LIN {X 0,Y 282.831,Z 361.895,A -85,B 0,C 180,E1 -17098.576,E2 -17098.576} C_VEL
LIN {X 0,Y 282.658,Z 360.951,A -85,B 0,C 180,E1 -17100,E2 -17100} C_VEL
LIN {X 0,Y 282.587,Z 359.569,A -85,B 0,C 180,E1 -17101.425,E2 -17101.425} C_VEL
LIN {X 0,Y 282.639,Z 356.738,A -85,B 0,C 180,E1 -17103.564,E2 -17103.564} C_VEL
LIN {X 0,Y 282.765,Z 351.895,A -85,B 0,C 180,E1 -17106.179,E2 -17106.179} C_VEL
LIN {X 0,Y 283.123,Z 346.036,A -85,B 0,C 180,E1 -17108.566,E2 -17108.566} C_VEL
LIN {X 0,Y 283.616,Z 339.368,A -85,B 0,C 180,E1 -17110.711,E2 -17110.711} C_VEL
LIN {X 0,Y 284.287,Z 331.159,A -85,B 0,C 180,E1 -17112.856,E2 -17112.856} C_VEL
LIN {X 0,Y 285.11,Z 322.916,A -85,B 0,C 180,E1 -17114.635,E2 -17114.635} C_VEL
LIN {X 0,Y 285.821,Z 314.704,A -85,B 0,C 180,E1 -17116.129,E2 -17116.129} C_VEL
LIN {X 0,Y 286.898,Z 303.457,A -85,B 0,C 180,E1 -17117.831,E2 -17117.831} C_VEL
LIN {X 0,Y 288.151,Z 290.351,A -85,B 0,C 180,E1 -17119.41,E2 -17119.41} C_VEL
LIN {X 0,Y 288.308,Z 286.867,A -85,B 0,C 180,E1 -17119.769,E2 -17119.769} C_VEL
LIN {X 0,Y 286.028,Z 274.318,A -85,B 0,C 180,E1 -17120.979,E2 -17120.979} C_VEL
LIN {X 0,Y 283.378,Z 259.454,A -85,B 0,C 180,E1 -17122.077,E2 -17122.077} C_VEL
LIN {X 0,Y 282.903,Z 256.645,A -85,B 0,C 180,E1 -17122.25,E2 -17122.25} C_VEL
LIN {X 0,Y 283.071,Z 253.228,A -85,B 0,C 180,E1 -17126.148,E2 -17126.148} C_VEL
LIN {X 0,Y 283.439,Z 253.178,A -85,B 0,C 180,E1 -17129.79,E2 -17129.79} C_VEL
LIN {X 0,Y 283.84,Z 253.128,A -85,B 0,C 180,E1 -17133.007,E2 -17133.007} C_VEL
LIN {X 0,Y 284.182,Z 253.083,A -85,B 0,C 180,E1 -17136.409,E2 -17136.409} C_VEL
LIN {X 0,Y 284.308,Z 253.067,A -85,B 0,C 180,E1 -17139.995,E2 -17139.995} C_VEL
LIN {X 0,Y 284.248,Z 253.076,A -85,B 0,C 180,E1 -17144.19,E2 -17144.19} C_VEL
LIN {X 0,Y 284.243,Z 253.076,A -85,B 0,C 180,E1 -17148.119,E2 -17148.119} C_VEL
LIN {X 0,Y 284.311,Z 253.069,A -85,B 0,C 180,E1 -17152.282,E2 -17152.282} C_VEL
LIN {X 0,Y 284.31,Z 253.069,A -85,B 0,C 180,E1 -17155.35,E2 -17155.35} C_VEL
LIN {X 0,Y 284.29,Z 253.074,A -85,B 0,C 180,E1 -17158.725,E2 -17158.725} C_VEL
LIN {X 0,Y 284.294,Z 253.071,A -85,B 0,C 180,E1 -17161.985,E2 -17161.985} C_VEL
LIN {X 0,Y 284.329,Z 253.068,A -85,B 0,C 180,E1 -17166.145,E2 -17166.145} C_VEL
LIN {X 0,Y 284.391,Z 253.059,A -85,B 0,C 180,E1 -17169.898,E2 -17169.898} C_VEL
LIN {X 0,Y 284.496,Z 253.047,A -85,B 0,C 180,E1 -17174.459,E2 -17174.459} C_VEL
LIN {X 0,Y 284.486,Z 253.048,A -85,B 0,C 180,E1 -17178.601,E2 -17178.601} C_VEL
LIN {X 0,Y 284.611,Z 253.033,A -85,B 0,C 180,E1 -17181.479,E2 -17181.479} C_VEL
LIN {X 0,Y 284.568,Z 253.038,A -85,B 0,C 180,E1 -17184.33,E2 -17184.33} C_VEL
LIN {X 0,Y 284.844,Z 253.003,A -85,B 0,C 180,E1 -17188.586,E2 -17188.586} C_VEL
LIN {X 0,Y 284.839,Z 253.007,A -85,B 0,C 180,E1 -17191.414,E2 -17191.414} C_VEL
LIN {X 0,Y 284.646,Z 253.052,A -85,B 0,C 180,E1 -17193.007,E2 -17193.007} C_VEL
LIN {X 0,Y 284.818,Z 258.793,A -85,B 0,C 180,E1 -17196.375,E2 -17196.375} C_VEL
LIN {X 0,Y 284.369,Z 266.259,A -85,B 0,C 180,E1 -17200.682,E2 -17200.682} C_VEL
LIN {X 0,Y 284.094,Z 272.577,A -85,B 0,C 180,E1 -17204.323,E2 -17204.323} C_VEL
LIN {X 0,Y 283.88,Z 279.623,A -85,B 0,C 180,E1 -17208.307,E2 -17208.307} C_VEL
LIN {X 0,Y 285.728,Z 289.55,A -85,B 0,C 180,E1 -17208.927,E2 -17208.927} C_VEL
LIN {X 0,Y 287.481,Z 300.318,A -85,B 0,C 180,E1 -17209.828,E2 -17209.828} C_VEL
LIN {X 0,Y 288.186,Z 306.947,A -85,B 0,C 180,E1 -17210.522,E2 -17210.522} C_VEL
LIN {X 0,Y 287.358,Z 316.725,A -85,B 0,C 180,E1 -17211.661,E2 -17211.661} C_VEL
LIN {X 0,Y 286.342,Z 326.267,A -85,B 0,C 180,E1 -17213.123,E2 -17213.123} C_VEL
LIN {X 0,Y 285.604,Z 333.152,A -85,B 0,C 180,E1 -17214.427,E2 -17214.427} C_VEL
LIN {X 0,Y 285.015,Z 338.231,A -85,B 0,C 180,E1 -17215.564,E2 -17215.564} C_VEL
LIN {X 0,Y 284.307,Z 344.063,A -85,B 0,C 180,E1 -17217.137,E2 -17217.137} C_VEL
LIN {X 0,Y 283.686,Z 349.285,A -85,B 0,C 180,E1 -17218.887,E2 -17218.887} C_VEL
LIN {X 0,Y 283.192,Z 353.281,A -85,B 0,C 180,E1 -17220.58,E2 -17220.58} C_VEL
LIN {X 0,Y 282.836,Z 356.48,A -85,B 0,C 180,E1 -17222.344,E2 -17222.344} C_VEL
LIN {X 0,Y 282.69,Z 357.695,A -85,B 0,C 180,E1 -17223.158,E2 -17223.158} C_VEL
LIN {X 0,Y 282.49,Z 359.603,A -85,B 0,C 180,E1 -17224.905,E2 -17224.905} C_VEL
LIN {X 0,Y 282.397,Z 360.883,A -85,B 0,C 180,E1 -17227.213,E2 -17227.213} C_VEL
LIN {X 0,Y 282.468,Z 361.102,A -85,B 0,C 180,E1 -17228.464,E2 -17228.464} C_VEL
LIN {X 0,Y 282.717,Z 360.662,A -85,B 0,C 180,E1 -17230.265,E2 -17230.265} C_VEL
LIN {X 0,Y 283.098,Z 359.387,A -85,B 0,C 180,E1 -17232.089,E2 -17232.089} C_VEL
LIN {X 0,Y 283.686,Z 356.998,A -85,B 0,C 180,E1 -17234.074,E2 -17234.074} C_VEL
LIN {X 0,Y 284.532,Z 353.138,A -85,B 0,C 180,E1 -17236.242,E2 -17236.242} C_VEL
LIN {X 0,Y 285.66,Z 347.925,A -85,B 0,C 180,E1 -17238.373,E2 -17238.373} C_VEL
LIN {X 0,Y 286.946,Z 340.998,A -85,B 0,C 180,E1 -17240.446,E2 -17240.446} C_VEL
LIN {X 0,Y 288.222,Z 334.615,A -85,B 0,C 180,E1 -17241.948,E2 -17241.948} C_VEL
LIN {X 0,Y 289.382,Z 327.787,A -85,B 0,C 180,E1 -17243.268,E2 -17243.268} C_VEL
LIN {X 0,Y 290.809,Z 318.256,A -85,B 0,C 180,E1 -17244.757,E2 -17244.757} C_VEL
LIN {X 0,Y 291.63,Z 311.075,A -85,B 0,C 180,E1 -17245.652,E2 -17245.652} C_VEL
LIN {X 0,Y 290.183,Z 300.685,A -85,B 0,C 180,E1 -17246.889,E2 -17246.889} C_VEL
LIN {X 0,Y 288.063,Z 291.312,A -85,B 0,C 180,E1 -17247.848,E2 -17247.848} C_VEL
LIN {X 0,Y 285.192,Z 281.882,A -85,B 0,C 180,E1 -17248.68,E2 -17248.68} C_VEL
LIN {X 0,Y 284.996,Z 280.806,A -85,B 0,C 180,E1 -17248.811,E2 -17248.811} C_VEL
LIN {X 0,Y 285.473,Z 273.627,A -85,B 0,C 180,E1 -17253.077,E2 -17253.077} C_VEL
LIN {X 0,Y 285.948,Z 266.001,A -85,B 0,C 180,E1 -17257.607,E2 -17257.607} C_VEL
LIN {X 0,Y 286.031,Z 262.289,A -85,B 0,C 180,E1 -17259.88,E2 -17259.88} C_VEL
LIN {X 0,Y 285.367,Z 257.623,A -85,B 0,C 180,E1 -17262.81,E2 -17262.81} C_VEL
LIN {X 0,Y 284.5,Z 253.05,A -85,B 0,C 180,E1 -17265.88,E2 -17265.88} C_VEL
LIN {X 0,Y 284.521,Z 253.047,A -85,B 0,C 180,E1 -17270.046,E2 -17270.046} C_VEL
LIN {X 0,Y 284.662,Z 253.027,A -85,B 0,C 180,E1 -17272.909,E2 -17272.909} C_VEL
LIN {X 0,Y 284.554,Z 253.037,A -85,B 0,C 180,E1 -17276.166,E2 -17276.166} C_VEL
LIN {X 0,Y 284.035,Z 253.105,A -85,B 0,C 180,E1 -17277.35,E2 -17277.35} C_VEL
LIN {X 0,Y 281.309,Z 253.443,A -85,B 0,C 180,E1 -17279.282,E2 -17279.282} C_VEL
LIN {X 0,Y 278.895,Z 253.747,A -85,B 0,C 180,E1 -17280.851,E2 -17280.851} C_VEL
LIN {X 0,Y 277.82,Z 253.879,A -85,B 0,C 180,E1 -17282.066,E2 -17282.066} C_VEL
LIN {X 0,Y 277.716,Z 253.89,A -85,B 0,C 180,E1 -17282.477,E2 -17282.477} C_VEL
LIN {X 0,Y 277.613,Z 253.907,A -85,B 0,C 180,E1 -17287.272,E2 -17287.272} C_VEL
LIN {X 0,Y 277.462,Z 253.924,A -85,B 0,C 180,E1 -17290.213,E2 -17290.213} C_VEL
LIN {X 0,Y 277.436,Z 253.928,A -85,B 0,C 180,E1 -17294.674,E2 -17294.674} C_VEL
LIN {X 0,Y 277.346,Z 253.935,A -85,B 0,C 180,E1 -17299.234,E2 -17299.234} C_VEL
LIN {X 0,Y 277.293,Z 253.941,A -85,B 0,C 180,E1 -17304.158,E2 -17304.158} C_VEL
LIN {X 0,Y 277.327,Z 253.938,A -85,B 0,C 180,E1 -17307.505,E2 -17307.505} C_VEL
LIN {X 0,Y 277.273,Z 253.947,A -85,B 0,C 180,E1 -17310.481,E2 -17310.481} C_VEL
LIN {X 0,Y 277.248,Z 253.949,A -85,B 0,C 180,E1 -17313.896,E2 -17313.896} C_VEL
LIN {X 0,Y 277.273,Z 253.943,A -85,B 0,C 180,E1 -17317.468,E2 -17317.468} C_VEL
LIN {X 0,Y 277.216,Z 253.954,A -85,B 0,C 180,E1 -17321.235,E2 -17321.235} C_VEL
LIN {X 0,Y 277.356,Z 254.102,A -85,B 0,C 180,E1 -17324.424,E2 -17324.424} C_VEL
LIN {X 0,Y 278.44,Z 259.918,A -85,B 0,C 180,E1 -17328.985,E2 -17328.985} C_VEL
LIN {X 0,Y 279.116,Z 264.08,A -85,B 0,C 180,E1 -17332.105,E2 -17332.105} C_VEL
LIN {X 0,Y 279.095,Z 267.562,A -85,B 0,C 180,E1 -17334.608,E2 -17334.608} C_VEL
LIN {X 0,Y 278.184,Z 272.378,A -85,B 0,C 180,E1 -17337.958,E2 -17337.958} C_VEL
LIN {X 0,Y 277.416,Z 277.12,A -85,B 0,C 180,E1 -17341.227,E2 -17341.227} C_VEL
LIN {X 0,Y 276.912,Z 281.064,A -85,B 0,C 180,E1 -17343.834,E2 -17343.834} C_VEL
LIN {X 0,Y 278.169,Z 295.048,A -85,B 0,C 180,E1 -17346.748,E2 -17346.748} C_VEL
LIN {X 0,Y 278.48,Z 299.439,A -85,B 0,C 180,E1 -17347.56,E2 -17347.56} C_VEL
LIN {X 0,Y 279.824,Z 307.988,A -85,B 0,C 180,E1 -17348.027,E2 -17348.027} C_VEL
LIN {X 0,Y 280.79,Z 317.875,A -85,B 0,C 180,E1 -17348.666,E2 -17348.666} C_VEL
LIN {X 0,Y 281.623,Z 328.142,A -85,B 0,C 180,E1 -17349.551,E2 -17349.551} C_VEL
LIN {X 0,Y 281.925,Z 335.562,A -85,B 0,C 180,E1 -17350.334,E2 -17350.334} C_VEL
LIN {X 0,Y 280.797,Z 346.088,A -85,B 0,C 180,E1 -17351.58,E2 -17351.58} C_VEL
LIN {X 0,Y 279.658,Z 354.16,A -85,B 0,C 180,E1 -17352.808,E2 -17352.808} C_VEL
LIN {X 0,Y 278.667,Z 361.864,A -85,B 0,C 180,E1 -17354.269,E2 -17354.269} C_VEL
LIN {X 0,Y 277.805,Z 368.163,A -85,B 0,C 180,E1 -17355.72,E2 -17355.72} C_VEL
LIN {X 0,Y 276.985,Z 373.425,A -85,B 0,C 180,E1 -17357.173,E2 -17357.173} C_VEL
LIN {X 0,Y 276.277,Z 378.801,A -85,B 0,C 180,E1 -17359.001,E2 -17359.001} C_VEL
LIN {X 0,Y 275.896,Z 382.288,A -85,B 0,C 180,E1 -17360.469,E2 -17360.469} C_VEL
LIN {X 0,Y 275.532,Z 386.34,A -85,B 0,C 180,E1 -17362.673,E2 -17362.673} C_VEL
LIN {X 0,Y 275.44,Z 388.507,A -85,B 0,C 180,E1 -17364.331,E2 -17364.331} C_VEL
LIN {X 0,Y 275.41,Z 389.721,A -85,B 0,C 180,E1 -17365.61,E2 -17365.61} C_VEL
LIN {X 0,Y 275.499,Z 390.664,A -85,B 0,C 180,E1 -17367.076,E2 -17367.076} C_VEL
LIN {X 0,Y 275.55,Z 391.055,A -85,B 0,C 180,E1 -17368.539,E2 -17368.539} C_VEL
LIN {X 0,Y 275.637,Z 390.67,A -85,B 0,C 180,E1 -17371.461,E2 -17371.461} C_VEL
LIN {X 0,Y 275.355,Z 391.344,A -85,B 0,C 180,E1 -17374.392,E2 -17374.392} C_VEL
LIN {X 0,Y 275.454,Z 390.474,A -85,B 0,C 180,E1 -17377.33,E2 -17377.33} C_VEL
LIN {X 0,Y 275.722,Z 389.465,A -85,B 0,C 180,E1 -17378.797,E2 -17378.797} C_VEL
LIN {X 0,Y 276.728,Z 386.251,A -85,B 0,C 180,E1 -17381.723,E2 -17381.723} C_VEL
LIN {X 0,Y 277.919,Z 382.837,A -85,B 0,C 180,E1 -17383.901,E2 -17383.901} C_VEL
LIN {X 0,Y 280.452,Z 376.813,A -85,B 0,C 180,E1 -17386.75,E2 -17386.75} C_VEL
LIN {X 0,Y 282.55,Z 371.143,A -85,B 0,C 180,E1 -17388.866,E2 -17388.866} C_VEL
LIN {X 0,Y 285.852,Z 363.067,A -85,B 0,C 180,E1 -17391.263,E2 -17391.263} C_VEL
LIN {X 0,Y 289.91,Z 353.174,A -85,B 0,C 180,E1 -17393.578,E2 -17393.578} C_VEL
LIN {X 0,Y 293.011,Z 344.832,A -85,B 0,C 180,E1 -17395.198,E2 -17395.198} C_VEL
LIN {X 0,Y 294.489,Z 337.714,A -85,B 0,C 180,E1 -17396.582,E2 -17396.582} C_VEL
LIN {X 0,Y 295.186,Z 329.455,A -85,B 0,C 180,E1 -17398.246,E2 -17398.246} C_VEL
LIN {X 0,Y 294.967,Z 319.929,A -85,B 0,C 180,E1 -17400.266,E2 -17400.266} C_VEL
LIN {X 0,Y 294.401,Z 313.67,A -85,B 0,C 180,E1 -17401.681,E2 -17401.681} C_VEL
LIN {X 0,Y 292.788,Z 303.44,A -85,B 0,C 180,E1 -17404.3,E2 -17404.3} C_VEL
LIN {X 0,Y 292.15,Z 300.019,A -85,B 0,C 180,E1 -17405.265,E2 -17405.265} C_VEL
LIN {X 0,Y 290.757,Z 294.362,A -85,B 0,C 180,E1 -17407.178,E2 -17407.178} C_VEL
LIN {X 0,Y 289.417,Z 289.757,A -85,B 0,C 180,E1 -17409.152,E2 -17409.152} C_VEL
LIN {X 0,Y 288.8,Z 287.91,A -85,B 0,C 180,E1 -17410.144,E2 -17410.144} C_VEL
LIN {X 0,Y 287.153,Z 284.531,A -85,B 0,C 180,E1 -17413.259,E2 -17413.259} C_VEL
LIN {X 0,Y 286.793,Z 283.133,A -85,B 0,C 180,E1 -17415.289,E2 -17415.289} C_VEL
LIN {X 0,Y 286.896,Z 282.566,A -85,B 0,C 180,E1 -17417.299,E2 -17417.299} C_VEL
LIN {X 0,Y 288.338,Z 282.932,A -85,B 0,C 180,E1 -17420.674,E2 -17420.674} C_VEL
LIN {X 0,Y 288.675,Z 283.13,A -85,B 0,C 180,E1 -17421.176,E2 -17421.176} C_VEL
LIN {X 0,Y 291.63,Z 287.665,A -85,B 0,C 180,E1 -17425.022,E2 -17425.022} C_VEL
LIN {X 0,Y 294.048,Z 292.584,A -85,B 0,C 180,E1 -17427.557,E2 -17427.557} C_VEL
LIN {X 0,Y 296.068,Z 297.264,A -85,B 0,C 180,E1 -17429.494,E2 -17429.494} C_VEL
LIN {X 0,Y 298.512,Z 305.114,A -85,B 0,C 180,E1 -17432.111,E2 -17432.111} C_VEL
LIN {X 0,Y 299.925,Z 313.163,A -85,B 0,C 180,E1 -17434.397,E2 -17434.397} C_VEL
LIN {X 0,Y 300.069,Z 314.428,A -85,B 0,C 180,E1 -17434.738,E2 -17434.738} C_VEL
LIN {X 0,Y 299.8,Z 315.956,A -85,B 0,C 180,E1 -17435.042,E2 -17435.042} C_VEL
LIN {X 0,Y 295.732,Z 326.426,A -85,B 0,C 180,E1 -17436.914,E2 -17436.914} C_VEL
LIN {X 0,Y 292.089,Z 335.102,A -85,B 0,C 180,E1 -17438.844,E2 -17438.844} C_VEL
LIN {X 0,Y 288.331,Z 343.318,A -85,B 0,C 180,E1 -17441.158,E2 -17441.158} C_VEL
LIN {X 0,Y 285.081,Z 349.926,A -85,B 0,C 180,E1 -17443.531,E2 -17443.531} C_VEL
LIN {X 0,Y 282.003,Z 355.656,A -85,B 0,C 180,E1 -17446.305,E2 -17446.305} C_VEL
LIN {X 0,Y 280.101,Z 358.853,A -85,B 0,C 180,E1 -17448.421,E2 -17448.421} C_VEL
LIN {X 0,Y 278.918,Z 360.509,A -85,B 0,C 180,E1 -17449.841,E2 -17449.841} C_VEL
LIN {X 0,Y 278.251,Z 361.729,A -85,B 0,C 180,E1 -17451.284,E2 -17451.284} C_VEL
LIN {X 0,Y 277.048,Z 363.021,A -85,B 0,C 180,E1 -17454.176,E2 -17454.176} C_VEL
LIN {X 0,Y 276.62,Z 363.112,A -85,B 0,C 180,E1 -17455.629,E2 -17455.629} C_VEL
LIN {X 0,Y 276.092,Z 362.846,A -85,B 0,C 180,E1 -17457.082,E2 -17457.082} C_VEL
LIN {X 0,Y 275.739,Z 362.169,A -85,B 0,C 180,E1 -17458.54,E2 -17458.54} C_VEL
LIN {X 0,Y 275.502,Z 359.588,A -85,B 0,C 180,E1 -17461.462,E2 -17461.462} C_VEL
LIN {X 0,Y 275.554,Z 356.575,A -85,B 0,C 180,E1 -17463.656,E2 -17463.656} C_VEL
LIN {X 0,Y 275.66,Z 352.015,A -85,B 0,C 180,E1 -17466.109,E2 -17466.109} C_VEL
LIN {X 0,Y 275.956,Z 347.388,A -85,B 0,C 180,E1 -17468.052,E2 -17468.052} C_VEL
LIN {X 0,Y 276.41,Z 340.976,A -85,B 0,C 180,E1 -17470.252,E2 -17470.252} C_VEL
LIN {X 0,Y 277.019,Z 333.069,A -85,B 0,C 180,E1 -17472.454,E2 -17472.454} C_VEL
LIN {X 0,Y 278,Z 323.322,A -85,B 0,C 180,E1 -17474.644,E2 -17474.644} C_VEL
LIN {X 0,Y 278.778,Z 314.188,A -85,B 0,C 180,E1 -17476.341,E2 -17476.341} C_VEL
LIN {X 0,Y 279.941,Z 302.606,A -85,B 0,C 180,E1 -17478.1,E2 -17478.1} C_VEL
LIN {X 0,Y 281.058,Z 290.91,A -85,B 0,C 180,E1 -17479.539,E2 -17479.539} C_VEL
LIN {X 0,Y 281.219,Z 287.457,A -85,B 0,C 180,E1 -17479.908,E2 -17479.908} C_VEL
LIN {X 0,Y 278.876,Z 274.615,A -85,B 0,C 180,E1 -17481.18,E2 -17481.18} C_VEL
LIN {X 0,Y 276.275,Z 259.963,A -85,B 0,C 180,E1 -17482.291,E2 -17482.291} C_VEL
LIN {X 0,Y 275.804,Z 257.028,A -85,B 0,C 180,E1 -17482.472,E2 -17482.472} C_VEL
LIN {X 0,Y 275.996,Z 254.109,A -85,B 0,C 180,E1 -17486.05,E2 -17486.05} C_VEL
LIN {X 0,Y 276.468,Z 254.045,A -85,B 0,C 180,E1 -17490.559,E2 -17490.559} C_VEL
LIN {X 0,Y 276.896,Z 253.99,A -85,B 0,C 180,E1 -17493.945,E2 -17493.945} C_VEL
LIN {X 0,Y 277.195,Z 253.957,A -85,B 0,C 180,E1 -17497.481,E2 -17497.481} C_VEL
LIN {X 0,Y 277.213,Z 253.955,A -85,B 0,C 180,E1 -17501.236,E2 -17501.236} C_VEL
LIN {X 0,Y 277.204,Z 253.956,A -85,B 0,C 180,E1 -17505.226,E2 -17505.226} C_VEL
LIN {X 0,Y 277.2,Z 253.955,A -85,B 0,C 180,E1 -17509.518,E2 -17509.518} C_VEL
LIN {X 0,Y 277.257,Z 253.949,A -85,B 0,C 180,E1 -17512.529,E2 -17512.529} C_VEL
LIN {X 0,Y 277.249,Z 253.949,A -85,B 0,C 180,E1 -17516.104,E2 -17516.104} C_VEL
LIN {X 0,Y 277.265,Z 253.945,A -85,B 0,C 180,E1 -17519.538,E2 -17519.538} C_VEL
LIN {X 0,Y 277.309,Z 253.942,A -85,B 0,C 180,E1 -17522.858,E2 -17522.858} C_VEL
LIN {X 0,Y 277.29,Z 253.944,A -85,B 0,C 180,E1 -17526.076,E2 -17526.076} C_VEL
LIN {X 0,Y 277.348,Z 253.935,A -85,B 0,C 180,E1 -17530.766,E2 -17530.766} C_VEL
LIN {X 0,Y 277.438,Z 253.924,A -85,B 0,C 180,E1 -17535.326,E2 -17535.326} C_VEL
LIN {X 0,Y 277.461,Z 253.925,A -85,B 0,C 180,E1 -17539.787,E2 -17539.787} C_VEL
LIN {X 0,Y 277.602,Z 253.905,A -85,B 0,C 180,E1 -17542.727,E2 -17542.727} C_VEL
LIN {X 0,Y 277.81,Z 253.879,A -85,B 0,C 180,E1 -17548.55,E2 -17548.55} C_VEL
LIN {X 0,Y 277.719,Z 253.892,A -85,B 0,C 180,E1 -17552.175,E2 -17552.175} C_VEL
LIN {X 0,Y 277.664,Z 254.036,A -85,B 0,C 180,E1 -17552.811,E2 -17552.811} C_VEL
LIN {X 0,Y 277.811,Z 259.03,A -85,B 0,C 180,E1 -17555.808,E2 -17555.808} C_VEL
LIN {X 0,Y 277.393,Z 266.586,A -85,B 0,C 180,E1 -17560.215,E2 -17560.215} C_VEL
LIN {X 0,Y 277.094,Z 272.975,A -85,B 0,C 180,E1 -17563.943,E2 -17563.943} C_VEL
LIN {X 0,Y 276.858,Z 279.85,A -85,B 0,C 180,E1 -17567.926,E2 -17567.926} C_VEL
LIN {X 0,Y 278.693,Z 289.804,A -85,B 0,C 180,E1 -17568.564,E2 -17568.564} C_VEL
LIN {X 0,Y 280.318,Z 299.627,A -85,B 0,C 180,E1 -17569.402,E2 -17569.402} C_VEL
LIN {X 0,Y 281.216,Z 306.242,A -85,B 0,C 180,E1 -17570.098,E2 -17570.098} C_VEL
LIN {X 0,Y 280.592,Z 314.904,A -85,B 0,C 180,E1 -17571.103,E2 -17571.103} C_VEL
LIN {X 0,Y 279.567,Z 324.771,A -85,B 0,C 180,E1 -17572.542,E2 -17572.542} C_VEL
LIN {X 0,Y 278.675,Z 332.941,A -85,B 0,C 180,E1 -17574.09,E2 -17574.09} C_VEL
LIN {X 0,Y 277.953,Z 338.903,A -85,B 0,C 180,E1 -17575.457,E2 -17575.457} C_VEL
LIN {X 0,Y 277.184,Z 344.955,A -85,B 0,C 180,E1 -17577.154,E2 -17577.154} C_VEL
LIN {X 0,Y 276.581,Z 349.874,A -85,B 0,C 180,E1 -17578.868,E2 -17578.868} C_VEL
LIN {X 0,Y 276.11,Z 353.826,A -85,B 0,C 180,E1 -17580.602,E2 -17580.602} C_VEL
LIN {X 0,Y 275.666,Z 357.483,A -85,B 0,C 180,E1 -17582.719,E2 -17582.719} C_VEL
LIN {X 0,Y 275.358,Z 360.186,A -85,B 0,C 180,E1 -17585.24,E2 -17585.24} C_VEL
LIN {X 0,Y 275.335,Z 361.392,A -85,B 0,C 180,E1 -17587.778,E2 -17587.778} C_VEL
LIN {X 0,Y 275.609,Z 361.227,A -85,B 0,C 180,E1 -17590.093,E2 -17590.093} C_VEL
LIN {X 0,Y 276.131,Z 359.671,A -85,B 0,C 180,E1 -17592.43,E2 -17592.43} C_VEL
LIN {X 0,Y 276.83,Z 356.888,A -85,B 0,C 180,E1 -17594.696,E2 -17594.696} C_VEL
LIN {X 0,Y 277.884,Z 352.329,A -85,B 0,C 180,E1 -17597.176,E2 -17597.176} C_VEL
LIN {X 0,Y 278.989,Z 347.362,A -85,B 0,C 180,E1 -17599.089,E2 -17599.089} C_VEL
LIN {X 0,Y 280.262,Z 340.907,A -85,B 0,C 180,E1 -17601.021,E2 -17601.021} C_VEL
LIN {X 0,Y 281.709,Z 333.87,A -85,B 0,C 180,E1 -17602.683,E2 -17602.683} C_VEL
LIN {X 0,Y 283.337,Z 324.577,A -85,B 0,C 180,E1 -17604.41,E2 -17604.41} C_VEL
LIN {X 0,Y 284.59,Z 316.244,A -85,B 0,C 180,E1 -17605.61,E2 -17605.61} C_VEL
LIN {X 0,Y 284.925,Z 311.04,A -85,B 0,C 180,E1 -17606.29,E2 -17606.29} C_VEL
LIN {X 0,Y 283.475,Z 301.24,A -85,B 0,C 180,E1 -17607.497,E2 -17607.497} C_VEL
LIN {X 0,Y 281.225,Z 291.571,A -85,B 0,C 180,E1 -17608.526,E2 -17608.526} C_VEL
LIN {X 0,Y 278.25,Z 281.865,A -85,B 0,C 180,E1 -17609.426,E2 -17609.426} C_VEL
LIN {X 0,Y 278.135,Z 281.189,A -85,B 0,C 180,E1 -17609.528,E2 -17609.528} C_VEL
LIN {X 0,Y 278.519,Z 275.466,A -85,B 0,C 180,E1 -17612.986,E2 -17612.986} C_VEL
LIN {X 0,Y 279.099,Z 267.527,A -85,B 0,C 180,E1 -17617.807,E2 -17617.807} C_VEL
LIN {X 0,Y 279.158,Z 263.819,A -85,B 0,C 180,E1 -17620.131,E2 -17620.131} C_VEL
LIN {X 0,Y 278.689,Z 260.323,A -85,B 0,C 180,E1 -17622.385,E2 -17622.385} C_VEL
LIN {X 0,Y 277.638,Z 254.834,A -85,B 0,C 180,E1 -17626.085,E2 -17626.085} C_VEL
LIN {X 0,Y 277.431,Z 253.926,A -85,B 0,C 180,E1 -17626.821,E2 -17626.821} C_VEL
LIN {X 0,Y 277.599,Z 253.908,A -85,B 0,C 180,E1 -17631.263,E2 -17631.263} C_VEL
LIN {X 0,Y 277.553,Z 253.912,A -85,B 0,C 180,E1 -17634.187,E2 -17634.187} C_VEL
LIN {X 0,Y 277.822,Z 253.88,A -85,B 0,C 180,E1 -17638.55,E2 -17638.55} C_VEL
LIN {X 0,Y 277.822,Z 253.877,A -85,B 0,C 180,E1 -17641.449,E2 -17641.449} C_VEL
LIN {X 0,Y 277.716,Z 253.89,A -85,B 0,C 180,E1 -17642.477,E2 -17642.477} C_VEL
LIN {X 0,Y 276.988,Z 253.984,A -85,B 0,C 180,E1 -17643.686,E2 -17643.686} C_VEL
LIN {X 0,Y 274.06,Z 254.346,A -85,B 0,C 180,E1 -17645.654,E2 -17645.654} C_VEL
LIN {X 0,Y 271.62,Z 254.653,A -85,B 0,C 180,E1 -17647.253,E2 -17647.253} C_VEL
LIN {X 0,Y 270.598,Z 254.776,A -85,B 0,C 180,E1 -17648.494,E2 -17648.494} C_VEL
LIN {X 0,Y 270.527,Z 254.786,A -85,B 0,C 180,E1 -17648.914,E2 -17648.914} C_VEL
LIN {X 0,Y 270.361,Z 254.804,A -85,B 0,C 180,E1 -17653.53,E2 -17653.53} C_VEL
LIN {X 0,Y 270.356,Z 254.805,A -85,B 0,C 180,E1 -17656.615,E2 -17656.615} C_VEL
LIN {X 0,Y 270.292,Z 254.816,A -85,B 0,C 180,E1 -17660.601,E2 -17660.601} C_VEL
LIN {X 0,Y 270.239,Z 254.821,A -85,B 0,C 180,E1 -17664.589,E2 -17664.589} C_VEL
LIN {X 0,Y 270.273,Z 254.82,A -85,B 0,C 180,E1 -17667.908,E2 -17667.908} C_VEL
LIN {X 0,Y 270.185,Z 254.828,A -85,B 0,C 180,E1 -17671.348,E2 -17671.348} C_VEL
LIN {X 0,Y 270.203,Z 254.823,A -85,B 0,C 180,E1 -17674.905,E2 -17674.905} C_VEL
LIN {X 0,Y 270.198,Z 254.828,A -85,B 0,C 180,E1 -17678.71,E2 -17678.71} C_VEL
LIN {X 0,Y 270.219,Z 254.827,A -85,B 0,C 180,E1 -17683.261,E2 -17683.261} C_VEL
LIN {X 0,Y 270.321,Z 255.015,A -85,B 0,C 180,E1 -17684.4,E2 -17684.4} C_VEL
LIN {X 0,Y 271.317,Z 260.334,A -85,B 0,C 180,E1 -17688.694,E2 -17688.694} C_VEL
LIN {X 0,Y 272.101,Z 265.284,A -85,B 0,C 180,E1 -17692.501,E2 -17692.501} C_VEL
LIN {X 0,Y 272.043,Z 267.943,A -85,B 0,C 180,E1 -17694.46,E2 -17694.46} C_VEL
LIN {X 0,Y 271.111,Z 272.74,A -85,B 0,C 180,E1 -17697.899,E2 -17697.899} C_VEL
LIN {X 0,Y 270.078,Z 279.195,A -85,B 0,C 180,E1 -17702.448,E2 -17702.448} C_VEL
LIN {X 0,Y 271.191,Z 292.709,A -85,B 0,C 180,E1 -17705.503,E2 -17705.503} C_VEL
LIN {X 0,Y 271.702,Z 299.153,A -85,B 0,C 180,E1 -17706.804,E2 -17706.804} C_VEL
LIN {X 0,Y 273.014,Z 305.084,A -85,B 0,C 180,E1 -17707.17,E2 -17707.17} C_VEL
LIN {X 0,Y 274.118,Z 316.132,A -85,B 0,C 180,E1 -17707.873,E2 -17707.873} C_VEL
LIN {X 0,Y 274.815,Z 324.964,A -85,B 0,C 180,E1 -17708.619,E2 -17708.619} C_VEL
LIN {X 0,Y 275.279,Z 332.949,A -85,B 0,C 180,E1 -17709.449,E2 -17709.449} C_VEL
LIN {X 0,Y 275.13,Z 338.107,A -85,B 0,C 180,E1 -17710.022,E2 -17710.022} C_VEL
LIN {X 0,Y 273.913,Z 347.731,A -85,B 0,C 180,E1 -17711.294,E2 -17711.294} C_VEL
LIN {X 0,Y 272.712,Z 355.5,A -85,B 0,C 180,E1 -17712.562,E2 -17712.562} C_VEL
LIN {X 0,Y 271.84,Z 362.018,A -85,B 0,C 180,E1 -17713.864,E2 -17713.864} C_VEL
LIN {X 0,Y 270.911,Z 368.227,A -85,B 0,C 180,E1 -17715.349,E2 -17715.349} C_VEL
LIN {X 0,Y 270.034,Z 373.41,A -85,B 0,C 180,E1 -17716.837,E2 -17716.837} C_VEL
LIN {X 0,Y 269.267,Z 378.717,A -85,B 0,C 180,E1 -17718.711,E2 -17718.711} C_VEL
LIN {X 0,Y 268.703,Z 383.684,A -85,B 0,C 180,E1 -17720.971,E2 -17720.971} C_VEL
LIN {X 0,Y 268.482,Z 386.126,A -85,B 0,C 180,E1 -17722.48,E2 -17722.48} C_VEL
LIN {X 0,Y 268.347,Z 388.481,A -85,B 0,C 180,E1 -17724.397,E2 -17724.397} C_VEL
LIN {X 0,Y 268.418,Z 390.298,A -85,B 0,C 180,E1 -17726.998,E2 -17726.998} C_VEL
LIN {X 0,Y 268.462,Z 390.675,A -85,B 0,C 180,E1 -17728.5,E2 -17728.5} C_VEL
LIN {X 0,Y 268.58,Z 390.182,A -85,B 0,C 180,E1 -17730.75,E2 -17730.75} C_VEL
LIN {X 0,Y 268.589,Z 389.936,A -85,B 0,C 180,E1 -17731.5,E2 -17731.5} C_VEL
LIN {X 0,Y 268.274,Z 390.848,A -85,B 0,C 180,E1 -17734.508,E2 -17734.508} C_VEL
LIN {X 0,Y 268.38,Z 390.158,A -85,B 0,C 180,E1 -17737.524,E2 -17737.524} C_VEL
LIN {X 0,Y 269.135,Z 387.986,A -85,B 0,C 180,E1 -17740.533,E2 -17740.533} C_VEL
LIN {X 0,Y 270.493,Z 384.273,A -85,B 0,C 180,E1 -17743.524,E2 -17743.524} C_VEL
LIN {X 0,Y 273.011,Z 378.971,A -85,B 0,C 180,E1 -17746.45,E2 -17746.45} C_VEL
LIN {X 0,Y 275.085,Z 373.902,A -85,B 0,C 180,E1 -17748.624,E2 -17748.624} C_VEL
LIN {X 0,Y 278.279,Z 366.688,A -85,B 0,C 180,E1 -17751.094,E2 -17751.094} C_VEL
LIN {X 0,Y 282.321,Z 357.765,A -85,B 0,C 180,E1 -17753.472,E2 -17753.472} C_VEL
LIN {X 0,Y 286.231,Z 348.637,A -85,B 0,C 180,E1 -17755.448,E2 -17755.448} C_VEL
LIN {X 0,Y 287.866,Z 343.658,A -85,B 0,C 180,E1 -17756.459,E2 -17756.459} C_VEL
LIN {X 0,Y 289.21,Z 336.008,A -85,B 0,C 180,E1 -17758.075,E2 -17758.075} C_VEL
LIN {X 0,Y 289.73,Z 328.434,A -85,B 0,C 180,E1 -17759.741,E2 -17759.741} C_VEL
LIN {X 0,Y 289.556,Z 319.516,A -85,B 0,C 180,E1 -17761.842,E2 -17761.842} C_VEL
LIN {X 0,Y 288.546,Z 308.938,A -85,B 0,C 180,E1 -17764.639,E2 -17764.639} C_VEL
LIN {X 0,Y 287.667,Z 303.831,A -85,B 0,C 180,E1 -17766.271,E2 -17766.271} C_VEL
LIN {X 0,Y 286.917,Z 299.667,A -85,B 0,C 180,E1 -17767.762,E2 -17767.762} C_VEL
LIN {X 0,Y 285.658,Z 294.321,A -85,B 0,C 180,E1 -17770.298,E2 -17770.298} C_VEL
LIN {X 0,Y 284.616,Z 292.114,A -85,B 0,C 180,E1 -17772.201,E2 -17772.201} C_VEL
LIN {X 0,Y 284.04,Z 290.41,A -85,B 0,C 180,E1 -17774.148,E2 -17774.148} C_VEL
LIN {X 0,Y 283.899,Z 289.365,A -85,B 0,C 180,E1 -17776.12,E2 -17776.12} C_VEL
LIN {X 0,Y 284.192,Z 289.048,A -85,B 0,C 180,E1 -17778.11,E2 -17778.11} C_VEL
LIN {X 0,Y 285.034,Z 289.279,A -85,B 0,C 180,E1 -17780.128,E2 -17780.128} C_VEL
LIN {X 0,Y 286.063,Z 290.648,A -85,B 0,C 180,E1 -17782.106,E2 -17782.106} C_VEL
LIN {X 0,Y 287.473,Z 292.73,A -85,B 0,C 180,E1 -17784.074,E2 -17784.074} C_VEL
LIN {X 0,Y 289.591,Z 297.026,A -85,B 0,C 180,E1 -17786.703,E2 -17786.703} C_VEL
LIN {X 0,Y 291.452,Z 302.054,A -85,B 0,C 180,E1 -17788.958,E2 -17788.958} C_VEL
LIN {X 0,Y 293.273,Z 308.654,A -85,B 0,C 180,E1 -17791.362,E2 -17791.362} C_VEL
LIN {X 0,Y 294.378,Z 315.987,A -85,B 0,C 180,E1 -17793.65,E2 -17793.65} C_VEL
LIN {X 0,Y 294.495,Z 317.575,A -85,B 0,C 180,E1 -17794.111,E2 -17794.111} C_VEL
LIN {X 0,Y 292.399,Z 323.083,A -85,B 0,C 180,E1 -17795.126,E2 -17795.126} C_VEL
LIN {X 0,Y 288.295,Z 332.38,A -85,B 0,C 180,E1 -17797.043,E2 -17797.043} C_VEL
LIN {X 0,Y 284.08,Z 341.169,A -85,B 0,C 180,E1 -17799.357,E2 -17799.357} C_VEL
LIN {X 0,Y 280.373,Z 348.284,A -85,B 0,C 180,E1 -17801.74,E2 -17801.74} C_VEL
LIN {X 0,Y 276.77,Z 354.558,A -85,B 0,C 180,E1 -17804.537,E2 -17804.537} C_VEL
LIN {X 0,Y 274.517,Z 358.134,A -85,B 0,C 180,E1 -17806.679,E2 -17806.679} C_VEL
LIN {X 0,Y 273.268,Z 360.015,A -85,B 0,C 180,E1 -17808.127,E2 -17808.127} C_VEL
LIN {X 0,Y 272.003,Z 361.516,A -85,B 0,C 180,E1 -17809.58,E2 -17809.58} C_VEL
LIN {X 0,Y 270.613,Z 363.273,A -85,B 0,C 180,E1 -17812.539,E2 -17812.539} C_VEL
LIN {X 0,Y 269.556,Z 363.604,A -85,B 0,C 180,E1 -17815.514,E2 -17815.514} C_VEL
LIN {X 0,Y 268.651,Z 362.367,A -85,B 0,C 180,E1 -17818.501,E2 -17818.501} C_VEL
LIN {X 0,Y 268.42,Z 359.585,A -85,B 0,C 180,E1 -17821.501,E2 -17821.501} C_VEL
LIN {X 0,Y 268.47,Z 356.387,A -85,B 0,C 180,E1 -17823.753,E2 -17823.753} C_VEL
LIN {X 0,Y 268.58,Z 351.997,A -85,B 0,C 180,E1 -17826.084,E2 -17826.084} C_VEL
LIN {X 0,Y 268.95,Z 345.751,A -85,B 0,C 180,E1 -17828.642,E2 -17828.642} C_VEL
LIN {X 0,Y 269.474,Z 338.853,A -85,B 0,C 180,E1 -17830.899,E2 -17830.899} C_VEL
LIN {X 0,Y 270.223,Z 330.396,A -85,B 0,C 180,E1 -17833.154,E2 -17833.154} C_VEL
LIN {X 0,Y 271.258,Z 319.93,A -85,B 0,C 180,E1 -17835.401,E2 -17835.401} C_VEL
LIN {X 0,Y 272.251,Z 309.547,A -85,B 0,C 180,E1 -17837.226,E2 -17837.226} C_VEL
LIN {X 0,Y 273.434,Z 297.458,A -85,B 0,C 180,E1 -17838.935,E2 -17838.935} C_VEL
LIN {X 0,Y 274.168,Z 289.673,A -85,B 0,C 180,E1 -17839.856,E2 -17839.856} C_VEL
LIN {X 0,Y 272.837,Z 280.584,A -85,B 0,C 180,E1 -17840.832,E2 -17840.832} C_VEL
LIN {X 0,Y 270.425,Z 267.286,A -85,B 0,C 180,E1 -17842.007,E2 -17842.007} C_VEL
LIN {X 0,Y 268.727,Z 257.374,A -85,B 0,C 180,E1 -17842.741,E2 -17842.741} C_VEL
LIN {X 0,Y 268.862,Z 254.997,A -85,B 0,C 180,E1 -17845.551,E2 -17845.551} C_VEL
LIN {X 0,Y 269.12,Z 254.965,A -85,B 0,C 180,E1 -17848.039,E2 -17848.039} C_VEL
LIN {X 0,Y 269.527,Z 254.914,A -85,B 0,C 180,E1 -17851.434,E2 -17851.434} C_VEL
LIN {X 0,Y 269.948,Z 254.857,A -85,B 0,C 180,E1 -17854.943,E2 -17854.943} C_VEL
LIN {X 0,Y 270.17,Z 254.831,A -85,B 0,C 180,E1 -17858.702,E2 -17858.702} C_VEL
LIN {X 0,Y 270.175,Z 254.829,A -85,B 0,C 180,E1 -17862.558,E2 -17862.558} C_VEL
LIN {X 0,Y 270.16,Z 254.834,A -85,B 0,C 180,E1 -17866.753,E2 -17866.753} C_VEL
LIN {X 0,Y 270.21,Z 254.826,A -85,B 0,C 180,E1 -17871.374,E2 -17871.374} C_VEL
LIN {X 0,Y 270.201,Z 254.828,A -85,B 0,C 180,E1 -17875.094,E2 -17875.094} C_VEL
LIN {X 0,Y 270.187,Z 254.828,A -85,B 0,C 180,E1 -17879.136,E2 -17879.136} C_VEL
LIN {X 0,Y 270.229,Z 254.824,A -85,B 0,C 180,E1 -17882.161,E2 -17882.161} C_VEL
LIN {X 0,Y 270.234,Z 254.821,A -85,B 0,C 180,E1 -17885.541,E2 -17885.541} C_VEL
LIN {X 0,Y 270.304,Z 254.817,A -85,B 0,C 180,E1 -17890.244,E2 -17890.244} C_VEL
LIN {X 0,Y 270.407,Z 254.8,A -85,B 0,C 180,E1 -17894.935,E2 -17894.935} C_VEL
LIN {X 0,Y 270.413,Z 254.801,A -85,B 0,C 180,E1 -17899.518,E2 -17899.518} C_VEL
LIN {X 0,Y 270.564,Z 254.782,A -85,B 0,C 180,E1 -17902.537,E2 -17902.537} C_VEL
LIN {X 0,Y 270.775,Z 254.756,A -85,B 0,C 180,E1 -17908.512,E2 -17908.512} C_VEL
LIN {X 0,Y 270.683,Z 254.806,A -85,B 0,C 180,E1 -17912.464,E2 -17912.464} C_VEL
LIN {X 0,Y 270.799,Z 260.562,A -85,B 0,C 180,E1 -17915.958,E2 -17915.958} C_VEL
LIN {X 0,Y 270.351,Z 268.152,A -85,B 0,C 180,E1 -17920.484,E2 -17920.484} C_VEL
LIN {X 0,Y 270.043,Z 274.642,A -85,B 0,C 180,E1 -17924.314,E2 -17924.314} C_VEL
LIN {X 0,Y 269.83,Z 280.123,A -85,B 0,C 180,E1 -17927.527,E2 -17927.527} C_VEL
LIN {X 0,Y 271.665,Z 290.066,A -85,B 0,C 180,E1 -17928.183,E2 -17928.183} C_VEL
LIN {X 0,Y 273.141,Z 298.975,A -85,B 0,C 180,E1 -17928.956,E2 -17928.956} C_VEL
LIN {X 0,Y 274.289,Z 307.272,A -85,B 0,C 180,E1 -17929.846,E2 -17929.846} C_VEL
LIN {X 0,Y 273.472,Z 317.445,A -85,B 0,C 180,E1 -17931.087,E2 -17931.087} C_VEL
LIN {X 0,Y 272.443,Z 326.582,A -85,B 0,C 180,E1 -17932.545,E2 -17932.545} C_VEL
LIN {X 0,Y 271.569,Z 334.166,A -85,B 0,C 180,E1 -17934.054,E2 -17934.054} C_VEL
LIN {X 0,Y 270.82,Z 340.097,A -85,B 0,C 180,E1 -17935.485,E2 -17935.485} C_VEL
LIN {X 0,Y 270.17,Z 345.161,A -85,B 0,C 180,E1 -17936.953,E2 -17936.953} C_VEL
LIN {X 0,Y 269.492,Z 350.461,A -85,B 0,C 180,E1 -17938.846,E2 -17938.846} C_VEL
LIN {X 0,Y 269.063,Z 354.039,A -85,B 0,C 180,E1 -17940.461,E2 -17940.461} C_VEL
LIN {X 0,Y 268.665,Z 357.248,A -85,B 0,C 180,E1 -17942.317,E2 -17942.317} C_VEL
LIN {X 0,Y 268.458,Z 358.661,A -85,B 0,C 180,E1 -17943.351,E2 -17943.351} C_VEL
LIN {X 0,Y 268.255,Z 360.837,A -85,B 0,C 180,E1 -17945.691,E2 -17945.691} C_VEL
LIN {X 0,Y 268.271,Z 361.857,A -85,B 0,C 180,E1 -17948.193,E2 -17948.193} C_VEL
LIN {X 0,Y 268.657,Z 361.341,A -85,B 0,C 180,E1 -17950.843,E2 -17950.843} C_VEL
LIN {X 0,Y 269.207,Z 359.717,A -85,B 0,C 180,E1 -17953.031,E2 -17953.031} C_VEL
LIN {X 0,Y 269.999,Z 356.8,A -85,B 0,C 180,E1 -17955.347,E2 -17955.347} C_VEL
LIN {X 0,Y 271.032,Z 352.627,A -85,B 0,C 180,E1 -17957.608,E2 -17957.608} C_VEL
LIN {X 0,Y 272.397,Z 346.815,A -85,B 0,C 180,E1 -17959.833,E2 -17959.833} C_VEL
LIN {X 0,Y 273.604,Z 341.014,A -85,B 0,C 180,E1 -17961.577,E2 -17961.577} C_VEL
LIN {X 0,Y 275.122,Z 333.944,A -85,B 0,C 180,E1 -17963.271,E2 -17963.271} C_VEL
LIN {X 0,Y 276.777,Z 324.896,A -85,B 0,C 180,E1 -17964.975,E2 -17964.975} C_VEL
LIN {X 0,Y 278.138,Z 316.329,A -85,B 0,C 180,E1 -17966.227,E2 -17966.227} C_VEL
LIN {X 0,Y 278.358,Z 312.583,A -85,B 0,C 180,E1 -17966.738,E2 -17966.738} C_VEL
LIN {X 0,Y 276.861,Z 302.262,A -85,B 0,C 180,E1 -17968.091,E2 -17968.091} C_VEL
LIN {X 0,Y 274.68,Z 292.772,A -85,B 0,C 180,E1 -17969.162,E2 -17969.162} C_VEL
LIN {X 0,Y 272.046,Z 284.157,A -85,B 0,C 180,E1 -17970.018,E2 -17970.018} C_VEL
LIN {X 0,Y 271.277,Z 281.652,A -85,B 0,C 180,E1 -17970.245,E2 -17970.245} C_VEL
LIN {X 0,Y 271.735,Z 275.699,A -85,B 0,C 180,E1 -17973.916,E2 -17973.916} C_VEL
LIN {X 0,Y 272.295,Z 268.606,A -85,B 0,C 180,E1 -17978.306,E2 -17978.306} C_VEL
LIN {X 0,Y 272.17,Z 264.182,A -85,B 0,C 180,E1 -17981.169,E2 -17981.169} C_VEL
LIN {X 0,Y 271.226,Z 258.555,A -85,B 0,C 180,E1 -17984.982,E2 -17984.982} C_VEL
LIN {X 0,Y 270.37,Z 254.81,A -85,B 0,C 180,E1 -17987.807,E2 -17987.807} C_VEL
LIN {X 0,Y 270.548,Z 254.786,A -85,B 0,C 180,E1 -17991.033,E2 -17991.033} C_VEL
LIN {X 0,Y 270.524,Z 254.787,A -85,B 0,C 180,E1 -17994.035,E2 -17994.035} C_VEL
LIN {X 0,Y 270.788,Z 254.757,A -85,B 0,C 180,E1 -17998.513,E2 -17998.513} C_VEL
LIN {X 0,Y 270.788,Z 254.754,A -85,B 0,C 180,E1 -18001.487,E2 -18001.487} C_VEL
LIN {X 0,Y 270.572,Z 254.783,A -85,B 0,C 180,E1 -18007.462,E2 -18007.462} C_VEL
LIN {X 0,Y 270.527,Z 254.786,A -85,B 0,C 180,E1 -18008.914,E2 -18008.914} C_VEL
LIN {X 0,Y 269.881,Z 254.872,A -85,B 0,C 180,E1 -18010.155,E2 -18010.155} C_VEL
LIN {X 0,Y 266.999,Z 255.236,A -85,B 0,C 180,E1 -18012.174,E2 -18012.174} C_VEL
LIN {X 0,Y 264.523,Z 255.541,A -85,B 0,C 180,E1 -18013.816,E2 -18013.816} C_VEL
LIN {X 0,Y 263.445,Z 255.67,A -85,B 0,C 180,E1 -18015.09,E2 -18015.09} C_VEL
LIN {X 0,Y 263.351,Z 255.679,A -85,B 0,C 180,E1 -18015.522,E2 -18015.522} C_VEL
LIN {X 0,Y 263.264,Z 255.693,A -85,B 0,C 180,E1 -18020.306,E2 -18020.306} C_VEL
LIN {X 0,Y 263.194,Z 255.702,A -85,B 0,C 180,E1 -18025.293,E2 -18025.293} C_VEL
LIN {X 0,Y 263.181,Z 255.701,A -85,B 0,C 180,E1 -18028.729,E2 -18028.729} C_VEL
LIN {X 0,Y 263.134,Z 255.704,A -85,B 0,C 180,E1 -18032.288,E2 -18032.288} C_VEL
LIN {X 0,Y 263.177,Z 255.703,A -85,B 0,C 180,E1 -18035.98,E2 -18035.98} C_VEL
LIN {X 0,Y 263.108,Z 255.708,A -85,B 0,C 180,E1 -18039.872,E2 -18039.872} C_VEL
LIN {X 0,Y 263.285,Z 255.712,A -85,B 0,C 180,E1 -18044.216,E2 -18044.216} C_VEL
LIN {X 0,Y 264.155,Z 260.635,A -85,B 0,C 180,E1 -18048.307,E2 -18048.307} C_VEL
LIN {X 0,Y 264.86,Z 264.543,A -85,B 0,C 180,E1 -18051.423,E2 -18051.423} C_VEL
LIN {X 0,Y 265.067,Z 267.257,A -85,B 0,C 180,E1 -18053.512,E2 -18053.512} C_VEL
LIN {X 0,Y 264.528,Z 270.696,A -85,B 0,C 180,E1 -18056.087,E2 -18056.087} C_VEL
LIN {X 0,Y 263.301,Z 277.443,A -85,B 0,C 180,E1 -18060.958,E2 -18060.958} C_VEL
LIN {X 0,Y 264.238,Z 289.01,A -85,B 0,C 180,E1 -18063.821,E2 -18063.821} C_VEL
LIN {X 0,Y 265.028,Z 299.062,A -85,B 0,C 180,E1 -18066.004,E2 -18066.004} C_VEL
LIN {X 0,Y 266.798,Z 306.615,A -85,B 0,C 180,E1 -18066.527,E2 -18066.527} C_VEL
LIN {X 0,Y 267.67,Z 316.522,A -85,B 0,C 180,E1 -18067.201,E2 -18067.201} C_VEL
LIN {X 0,Y 268.264,Z 325.652,A -85,B 0,C 180,E1 -18068.014,E2 -18068.014} C_VEL
LIN {X 0,Y 268.751,Z 335.626,A -85,B 0,C 180,E1 -18069.127,E2 -18069.127} C_VEL
LIN {X 0,Y 267.609,Z 345.827,A -85,B 0,C 180,E1 -18070.437,E2 -18070.437} C_VEL
LIN {X 0,Y 266.144,Z 354.866,A -85,B 0,C 180,E1 -18071.924,E2 -18071.924} C_VEL
LIN {X 0,Y 265.265,Z 360.547,A -85,B 0,C 180,E1 -18073.056,E2 -18073.056} C_VEL
LIN {X 0,Y 264.25,Z 366.91,A -85,B 0,C 180,E1 -18074.576,E2 -18074.576} C_VEL
LIN {X 0,Y 263.1,Z 373.409,A -85,B 0,C 180,E1 -18076.483,E2 -18076.483} C_VEL
LIN {X 0,Y 262.273,Z 378.636,A -85,B 0,C 180,E1 -18078.406,E2 -18078.406} C_VEL
LIN {X 0,Y 261.671,Z 383.516,A -85,B 0,C 180,E1 -18080.727,E2 -18080.727} C_VEL
LIN {X 0,Y 261.402,Z 385.922,A -85,B 0,C 180,E1 -18082.275,E2 -18082.275} C_VEL
LIN {X 0,Y 261.244,Z 388.466,A -85,B 0,C 180,E1 -18084.489,E2 -18084.489} C_VEL
LIN {X 0,Y 261.338,Z 389.934,A -85,B 0,C 180,E1 -18086.917,E2 -18086.917} C_VEL
LIN {X 0,Y 261.377,Z 390.283,A -85,B 0,C 180,E1 -18088.459,E2 -18088.459} C_VEL
LIN {X 0,Y 261.515,Z 390.047,A -85,B 0,C 180,E1 -18090,E2 -18090} C_VEL
LIN {X 0,Y 261.491,Z 389.285,A -85,B 0,C 180,E1 -18091.733,E2 -18091.733} C_VEL
LIN {X 0,Y 261.196,Z 390.278,A -85,B 0,C 180,E1 -18094.63,E2 -18094.63} C_VEL
LIN {X 0,Y 261.321,Z 389.847,A -85,B 0,C 180,E1 -18097.728,E2 -18097.728} C_VEL
LIN {X 0,Y 262.116,Z 387.879,A -85,B 0,C 180,E1 -18100.818,E2 -18100.818} C_VEL
LIN {X 0,Y 263.588,Z 384.458,A -85,B 0,C 180,E1 -18103.885,E2 -18103.885} C_VEL
LIN {X 0,Y 265.496,Z 380.85,A -85,B 0,C 180,E1 -18106.138,E2 -18106.138} C_VEL
LIN {X 0,Y 267.606,Z 376.358,A -85,B 0,C 180,E1 -18108.37,E2 -18108.37} C_VEL
LIN {X 0,Y 270.638,Z 370.013,A -85,B 0,C 180,E1 -18110.881,E2 -18110.881} C_VEL
LIN {X 0,Y 274.695,Z 361.939,A -85,B 0,C 180,E1 -18113.364,E2 -18113.364} C_VEL
LIN {X 0,Y 279.346,Z 352.231,A -85,B 0,C 180,E1 -18115.721,E2 -18115.721} C_VEL
LIN {X 0,Y 281.858,Z 345.945,A -85,B 0,C 180,E1 -18117.069,E2 -18117.069} C_VEL
LIN {X 0,Y 283.635,Z 337.61,A -85,B 0,C 180,E1 -18118.962,E2 -18118.962} C_VEL
LIN {X 0,Y 284.351,Z 329.685,A -85,B 0,C 180,E1 -18120.854,E2 -18120.854} C_VEL
LIN {X 0,Y 284.414,Z 321.587,A -85,B 0,C 180,E1 -18122.932,E2 -18122.932} C_VEL
LIN {X 0,Y 283.927,Z 312.738,A -85,B 0,C 180,E1 -18125.503,E2 -18125.503} C_VEL
LIN {X 0,Y 283.207,Z 305.963,A -85,B 0,C 180,E1 -18127.869,E2 -18127.869} C_VEL
LIN {X 0,Y 282.294,Z 300.779,A -85,B 0,C 180,E1 -18130.339,E2 -18130.339} C_VEL
LIN {X 0,Y 281.352,Z 298.326,A -85,B 0,C 180,E1 -18132.412,E2 -18132.412} C_VEL
LIN {X 0,Y 280.787,Z 296.029,A -85,B 0,C 180,E1 -18135.506,E2 -18135.506} C_VEL
LIN {X 0,Y 281.193,Z 295.444,A -85,B 0,C 180,E1 -18138.574,E2 -18138.574} C_VEL
LIN {X 0,Y 281.995,Z 295.896,A -85,B 0,C 180,E1 -18140.588,E2 -18140.588} C_VEL
LIN {X 0,Y 282.982,Z 297.458,A -85,B 0,C 180,E1 -18142.631,E2 -18142.631} C_VEL
LIN {X 0,Y 284.291,Z 299.78,A -85,B 0,C 180,E1 -18144.667,E2 -18144.667} C_VEL
LIN {X 0,Y 285.685,Z 303.317,A -85,B 0,C 180,E1 -18146.765,E2 -18146.765} C_VEL
LIN {X 0,Y 287.157,Z 308.356,A -85,B 0,C 180,E1 -18149.072,E2 -18149.072} C_VEL
LIN {X 0,Y 288.387,Z 314.258,A -85,B 0,C 180,E1 -18151.322,E2 -18151.322} C_VEL
LIN {X 0,Y 288.939,Z 320.515,A -85,B 0,C 180,E1 -18153.39,E2 -18153.39} C_VEL
LIN {X 0,Y 287.159,Z 324.891,A -85,B 0,C 180,E1 -18154.252,E2 -18154.252} C_VEL
LIN {X 0,Y 282.822,Z 333.869,A -85,B 0,C 180,E1 -18156.184,E2 -18156.184} C_VEL
LIN {X 0,Y 278.35,Z 342.444,A -85,B 0,C 180,E1 -18158.524,E2 -18158.524} C_VEL
LIN {X 0,Y 274.921,Z 348.468,A -85,B 0,C 180,E1 -18160.59,E2 -18160.59} C_VEL
LIN {X 0,Y 270.972,Z 354.784,A -85,B 0,C 180,E1 -18163.423,E2 -18163.423} C_VEL
LIN {X 0,Y 268.472,Z 358.412,A -85,B 0,C 180,E1 -18165.601,E2 -18165.601} C_VEL
LIN {X 0,Y 266.413,Z 361.126,A -85,B 0,C 180,E1 -18167.817,E2 -18167.817} C_VEL
LIN {X 0,Y 265.088,Z 362.475,A -85,B 0,C 180,E1 -18169.305,E2 -18169.305} C_VEL
LIN {X 0,Y 263.623,Z 363.99,A -85,B 0,C 180,E1 -18172.34,E2 -18172.34} C_VEL
LIN {X 0,Y 262.488,Z 364.009,A -85,B 0,C 180,E1 -18175.393,E2 -18175.393} C_VEL
LIN {X 0,Y 261.565,Z 362.551,A -85,B 0,C 180,E1 -18178.461,E2 -18178.461} C_VEL
LIN {X 0,Y 261.391,Z 361.228,A -85,B 0,C 180,E1 -18180,E2 -18180} C_VEL
LIN {X 0,Y 261.382,Z 357.333,A -85,B 0,C 180,E1 -18183.083,E2 -18183.083} C_VEL
LIN {X 0,Y 261.411,Z 353.325,A -85,B 0,C 180,E1 -18185.361,E2 -18185.361} C_VEL
LIN {X 0,Y 261.772,Z 347.105,A -85,B 0,C 180,E1 -18188.103,E2 -18188.103} C_VEL
LIN {X 0,Y 262.252,Z 340.399,A -85,B 0,C 180,E1 -18190.422,E2 -18190.422} C_VEL
LIN {X 0,Y 262.913,Z 332.173,A -85,B 0,C 180,E1 -18192.741,E2 -18192.741} C_VEL
LIN {X 0,Y 263.796,Z 323.95,A -85,B 0,C 180,E1 -18194.661,E2 -18194.661} C_VEL
LIN {X 0,Y 264.66,Z 314.045,A -85,B 0,C 180,E1 -18196.587,E2 -18196.587} C_VEL
LIN {X 0,Y 265.911,Z 301.924,A -85,B 0,C 180,E1 -18198.491,E2 -18198.491} C_VEL
LIN {X 0,Y 267.1,Z 289.958,A -85,B 0,C 180,E1 -18200.003,E2 -18200.003} C_VEL
LIN {X 0,Y 265.285,Z 278.979,A -85,B 0,C 180,E1 -18201.193,E2 -18201.193} C_VEL
LIN {X 0,Y 263.058,Z 266.205,A -85,B 0,C 180,E1 -18202.321,E2 -18202.321} C_VEL
LIN {X 0,Y 261.666,Z 257.79,A -85,B 0,C 180,E1 -18202.921,E2 -18202.921} C_VEL
LIN {X 0,Y 261.804,Z 255.876,A -85,B 0,C 180,E1 -18205.437,E2 -18205.437} C_VEL
LIN {X 0,Y 262.152,Z 255.83,A -85,B 0,C 180,E1 -18208.853,E2 -18208.853} C_VEL
LIN {X 0,Y 262.591,Z 255.773,A -85,B 0,C 180,E1 -18212.363,E2 -18212.363} C_VEL
LIN {X 0,Y 262.98,Z 255.725,A -85,B 0,C 180,E1 -18216.011,E2 -18216.011} C_VEL
LIN {X 0,Y 263.1,Z 255.71,A -85,B 0,C 180,E1 -18219.874,E2 -18219.874} C_VEL
LIN {X 0,Y 263.107,Z 255.71,A -85,B 0,C 180,E1 -18223.988,E2 -18223.988} C_VEL
LIN {X 0,Y 263.112,Z 255.709,A -85,B 0,C 180,E1 -18228.41,E2 -18228.41} C_VEL
LIN {X 0,Y 263.16,Z 255.703,A -85,B 0,C 180,E1 -18232.102,E2 -18232.102} C_VEL
LIN {X 0,Y 263.154,Z 255.704,A -85,B 0,C 180,E1 -18235.885,E2 -18235.885} C_VEL
LIN {X 0,Y 263.13,Z 255.706,A -85,B 0,C 180,E1 -18239.504,E2 -18239.504} C_VEL
LIN {X 0,Y 263.157,Z 255.704,A -85,B 0,C 180,E1 -18242.998,E2 -18242.998} C_VEL
LIN {X 0,Y 263.153,Z 255.707,A -85,B 0,C 180,E1 -18246.384,E2 -18246.384} C_VEL
LIN {X 0,Y 263.266,Z 255.69,A -85,B 0,C 180,E1 -18249.693,E2 -18249.693} C_VEL
LIN {X 0,Y 263.354,Z 255.681,A -85,B 0,C 180,E1 -18254.522,E2 -18254.522} C_VEL
LIN {X 0,Y 263.356,Z 255.679,A -85,B 0,C 180,E1 -18259.233,E2 -18259.233} C_VEL
LIN {X 0,Y 263.528,Z 255.66,A -85,B 0,C 180,E1 -18262.337,E2 -18262.337} C_VEL
LIN {X 0,Y 263.738,Z 255.633,A -85,B 0,C 180,E1 -18268.473,E2 -18268.473} C_VEL
LIN {X 0,Y 263.68,Z 255.712,A -85,B 0,C 180,E1 -18272.196,E2 -18272.196} C_VEL
LIN {X 0,Y 263.814,Z 260.847,A -85,B 0,C 180,E1 -18275.35,E2 -18275.35} C_VEL
LIN {X 0,Y 263.447,Z 267.219,A -85,B 0,C 180,E1 -18279.228,E2 -18279.228} C_VEL
LIN {X 0,Y 263.108,Z 273.687,A -85,B 0,C 180,E1 -18283.123,E2 -18283.123} C_VEL
LIN {X 0,Y 262.846,Z 280.357,A -85,B 0,C 180,E1 -18287.105,E2 -18287.105} C_VEL
LIN {X 0,Y 264.838,Z 291.333,A -85,B 0,C 180,E1 -18287.868,E2 -18287.868} C_VEL
LIN {X 0,Y 266.557,Z 301.941,A -85,B 0,C 180,E1 -18288.843,E2 -18288.843} C_VEL
LIN {X 0,Y 267.374,Z 308.296,A -85,B 0,C 180,E1 -18289.581,E2 -18289.581} C_VEL
LIN {X 0,Y 266.487,Z 318.34,A -85,B 0,C 180,E1 -18290.857,E2 -18290.857} C_VEL
LIN {X 0,Y 265.427,Z 327.279,A -85,B 0,C 180,E1 -18292.336,E2 -18292.336} C_VEL
LIN {X 0,Y 264.542,Z 334.879,A -85,B 0,C 180,E1 -18293.9,E2 -18293.9} C_VEL
LIN {X 0,Y 263.647,Z 341.861,A -85,B 0,C 180,E1 -18295.669,E2 -18295.669} C_VEL
LIN {X 0,Y 262.664,Z 348.991,A -85,B 0,C 180,E1 -18297.997,E2 -18297.997} C_VEL
LIN {X 0,Y 262.154,Z 353.099,A -85,B 0,C 180,E1 -18299.733,E2 -18299.733} C_VEL
LIN {X 0,Y 261.7,Z 356.567,A -85,B 0,C 180,E1 -18301.603,E2 -18301.603} C_VEL
LIN {X 0,Y 261.339,Z 359.21,A -85,B 0,C 180,E1 -18303.523,E2 -18303.523} C_VEL
LIN {X 0,Y 261.151,Z 361.571,A -85,B 0,C 180,E1 -18306.303,E2 -18306.303} C_VEL
LIN {X 0,Y 261.259,Z 362.301,A -85,B 0,C 180,E1 -18308.728,E2 -18308.728} C_VEL
LIN {X 0,Y 261.654,Z 361.65,A -85,B 0,C 180,E1 -18311.229,E2 -18311.229} C_VEL
LIN {X 0,Y 262.313,Z 359.779,A -85,B 0,C 180,E1 -18313.664,E2 -18313.664} C_VEL
LIN {X 0,Y 263.263,Z 356.59,A -85,B 0,C 180,E1 -18316.119,E2 -18316.119} C_VEL
LIN {X 0,Y 264.575,Z 351.412,A -85,B 0,C 180,E1 -18318.696,E2 -18318.696} C_VEL
LIN {X 0,Y 265.501,Z 347.67,A -85,B 0,C 180,E1 -18320.143,E2 -18320.143} C_VEL
LIN {X 0,Y 266.641,Z 342.632,A -85,B 0,C 180,E1 -18321.743,E2 -18321.743} C_VEL
LIN {X 0,Y 268.155,Z 336.034,A -85,B 0,C 180,E1 -18323.425,E2 -18323.425} C_VEL
LIN {X 0,Y 269.568,Z 329.068,A -85,B 0,C 180,E1 -18324.875,E2 -18324.875} C_VEL
LIN {X 0,Y 271.209,Z 319.96,A -85,B 0,C 180,E1 -18326.403,E2 -18326.403} C_VEL
LIN {X 0,Y 271.845,Z 314.75,A -85,B 0,C 180,E1 -18327.118,E2 -18327.118} C_VEL
LIN {X 0,Y 270.637,Z 305.119,A -85,B 0,C 180,E1 -18328.492,E2 -18328.492} C_VEL
LIN {X 0,Y 268.221,Z 294.065,A -85,B 0,C 180,E1 -18329.817,E2 -18329.817} C_VEL
LIN {X 0,Y 265.27,Z 284.643,A -85,B 0,C 180,E1 -18330.813,E2 -18330.813} C_VEL
LIN {X 0,Y 264.446,Z 281.98,A -85,B 0,C 180,E1 -18331.095,E2 -18331.095} C_VEL
LIN {X 0,Y 264.925,Z 275.973,A -85,B 0,C 180,E1 -18334.884,E2 -18334.884} C_VEL
LIN {X 0,Y 265.522,Z 269.396,A -85,B 0,C 180,E1 -18339.064,E2 -18339.064} C_VEL
LIN {X 0,Y 265.313,Z 265.825,A -85,B 0,C 180,E1 -18341.465,E2 -18341.465} C_VEL
LIN {X 0,Y 264.407,Z 260.304,A -85,B 0,C 180,E1 -18345.374,E2 -18345.374} C_VEL
LIN {X 0,Y 263.355,Z 255.684,A -85,B 0,C 180,E1 -18348.844,E2 -18348.844} C_VEL
LIN {X 0,Y 263.546,Z 255.658,A -85,B 0,C 180,E1 -18352.337,E2 -18352.337} C_VEL
LIN {X 0,Y 263.752,Z 255.633,A -85,B 0,C 180,E1 -18358.473,E2 -18358.473} C_VEL
LIN {X 0,Y 263.752,Z 255.63,A -85,B 0,C 180,E1 -18361.527,E2 -18361.527} C_VEL
LIN {X 0,Y 263.534,Z 255.659,A -85,B 0,C 180,E1 -18367.663,E2 -18367.663} C_VEL
LIN {X 0,Y 263.356,Z 255.677,A -85,B 0,C 180,E1 -18370.766,E2 -18370.766} C_VEL
LIN {X 0,Y 263.351,Z 255.679,A -85,B 0,C 180,E1 -18375.522,E2 -18375.522} C_VEL
LIN {X 0,Y 262.647,Z 255.768,A -85,B 0,C 180,E1 -18376.797,E2 -18376.797} C_VEL
LIN {X 0,Y 259.716,Z 256.13,A -85,B 0,C 180,E1 -18378.873,E2 -18378.873} C_VEL
LIN {X 0,Y 257.237,Z 256.442,A -85,B 0,C 180,E1 -18380.561,E2 -18380.561} C_VEL
LIN {X 0,Y 256.172,Z 256.572,A -85,B 0,C 180,E1 -18381.872,E2 -18381.872} C_VEL
LIN {X 0,Y 256.085,Z 256.585,A -85,B 0,C 180,E1 -18382.317,E2 -18382.317} C_VEL
LIN {X 0,Y 256.131,Z 256.579,A -85,B 0,C 180,E1 -18386.042,E2 -18386.042} C_VEL
LIN {X 0,Y 256.115,Z 256.578,A -85,B 0,C 180,E1 -18389.599,E2 -18389.599} C_VEL
LIN {X 0,Y 256.077,Z 256.587,A -85,B 0,C 180,E1 -18393.291,E2 -18393.291} C_VEL
LIN {X 0,Y 256.123,Z 256.577,A -85,B 0,C 180,E1 -18397.273,E2 -18397.273} C_VEL
LIN {X 0,Y 256.111,Z 256.58,A -85,B 0,C 180,E1 -18402.191,E2 -18402.191} C_VEL
LIN {X 0,Y 256.253,Z 256.589,A -85,B 0,C 180,E1 -18404.212,E2 -18404.212} C_VEL
LIN {X 0,Y 257.261,Z 262.269,A -85,B 0,C 180,E1 -18409.031,E2 -18409.031} C_VEL
LIN {X 0,Y 257.926,Z 266.159,A -85,B 0,C 180,E1 -18412.204,E2 -18412.204} C_VEL
LIN {X 0,Y 257.746,Z 269.608,A -85,B 0,C 180,E1 -18414.887,E2 -18414.887} C_VEL
LIN {X 0,Y 256.588,Z 275.31,A -85,B 0,C 180,E1 -18419.213,E2 -18419.213} C_VEL
LIN {X 0,Y 257.638,Z 288.904,A -85,B 0,C 180,E1 -18422.856,E2 -18422.856} C_VEL
LIN {X 0,Y 258.24,Z 298.702,A -85,B 0,C 180,E1 -18425.126,E2 -18425.126} C_VEL
LIN {X 0,Y 260.643,Z 308.277,A -85,B 0,C 180,E1 -18425.862,E2 -18425.862} C_VEL
LIN {X 0,Y 261.408,Z 318.592,A -85,B 0,C 180,E1 -18426.623,E2 -18426.623} C_VEL
LIN {X 0,Y 262.015,Z 330.313,A -85,B 0,C 180,E1 -18427.806,E2 -18427.806} C_VEL
LIN {X 0,Y 262.12,Z 338.098,A -85,B 0,C 180,E1 -18428.779,E2 -18428.779} C_VEL
LIN {X 0,Y 260.757,Z 347.536,A -85,B 0,C 180,E1 -18430.107,E2 -18430.107} C_VEL
LIN {X 0,Y 259.354,Z 355.637,A -85,B 0,C 180,E1 -18431.52,E2 -18431.52} C_VEL
LIN {X 0,Y 258.474,Z 360.771,A -85,B 0,C 180,E1 -18432.597,E2 -18432.597} C_VEL
LIN {X 0,Y 257.402,Z 367.032,A -85,B 0,C 180,E1 -18434.155,E2 -18434.155} C_VEL
LIN {X 0,Y 256.443,Z 372.266,A -85,B 0,C 180,E1 -18435.721,E2 -18435.721} C_VEL
LIN {X 0,Y 255.558,Z 376.654,A -85,B 0,C 180,E1 -18437.291,E2 -18437.291} C_VEL
LIN {X 0,Y 254.788,Z 381.867,A -85,B 0,C 180,E1 -18439.672,E2 -18439.672} C_VEL
LIN {X 0,Y 254.345,Z 385.722,A -85,B 0,C 180,E1 -18442.059,E2 -18442.059} C_VEL
LIN {X 0,Y 254.144,Z 388.341,A -85,B 0,C 180,E1 -18444.582,E2 -18444.582} C_VEL
LIN {X 0,Y 254.237,Z 389.57,A -85,B 0,C 180,E1 -18446.831,E2 -18446.831} C_VEL
LIN {X 0,Y 254.294,Z 389.878,A -85,B 0,C 180,E1 -18448.417,E2 -18448.417} C_VEL
LIN {X 0,Y 254.425,Z 389.63,A -85,B 0,C 180,E1 -18450,E2 -18450} C_VEL
LIN {X 0,Y 254.402,Z 388.619,A -85,B 0,C 180,E1 -18451.979,E2 -18451.979} C_VEL
LIN {X 0,Y 254.086,Z 389.748,A -85,B 0,C 180,E1 -18455.278,E2 -18455.278} C_VEL
LIN {X 0,Y 254.283,Z 389.466,A -85,B 0,C 180,E1 -18457.944,E2 -18457.944} C_VEL
LIN {X 0,Y 255.112,Z 387.786,A -85,B 0,C 180,E1 -18461.119,E2 -18461.119} C_VEL
LIN {X 0,Y 256.701,Z 384.603,A -85,B 0,C 180,E1 -18464.265,E2 -18464.265} C_VEL
LIN {X 0,Y 259.448,Z 379.94,A -85,B 0,C 180,E1 -18467.336,E2 -18467.336} C_VEL
LIN {X 0,Y 261.772,Z 375.402,A -85,B 0,C 180,E1 -18469.609,E2 -18469.609} C_VEL
LIN {X 0,Y 265.267,Z 368.923,A -85,B 0,C 180,E1 -18472.182,E2 -18472.182} C_VEL
LIN {X 0,Y 269.629,Z 360.913,A -85,B 0,C 180,E1 -18474.649,E2 -18474.649} C_VEL
LIN {X 0,Y 274.604,Z 351.25,A -85,B 0,C 180,E1 -18477.019,E2 -18477.019} C_VEL
LIN {X 0,Y 276.402,Z 346.723,A -85,B 0,C 180,E1 -18478.06,E2 -18478.06} C_VEL
LIN {X 0,Y 278.127,Z 339.229,A -85,B 0,C 180,E1 -18479.895,E2 -18479.895} C_VEL
LIN {X 0,Y 279.081,Z 331.407,A -85,B 0,C 180,E1 -18481.927,E2 -18481.927} C_VEL
LIN {X 0,Y 279.37,Z 323.534,A -85,B 0,C 180,E1 -18484.16,E2 -18484.16} C_VEL
LIN {X 0,Y 279.323,Z 315.457,A -85,B 0,C 180,E1 -18486.734,E2 -18486.734} C_VEL
LIN {X 0,Y 278.985,Z 310.604,A -85,B 0,C 180,E1 -18488.654,E2 -18488.654} C_VEL
LIN {X 0,Y 278.392,Z 306.149,A -85,B 0,C 180,E1 -18491.024,E2 -18491.024} C_VEL
LIN {X 0,Y 277.705,Z 303.967,A -85,B 0,C 180,E1 -18493.103,E2 -18493.103} C_VEL
LIN {X 0,Y 277.409,Z 302.483,A -85,B 0,C 180,E1 -18495.184,E2 -18495.184} C_VEL
LIN {X 0,Y 277.501,Z 301.77,A -85,B 0,C 180,E1 -18497.262,E2 -18497.262} C_VEL
LIN {X 0,Y 278.016,Z 301.706,A -85,B 0,C 180,E1 -18499.322,E2 -18499.322} C_VEL
LIN {X 0,Y 278.82,Z 302.519,A -85,B 0,C 180,E1 -18501.389,E2 -18501.389} C_VEL
LIN {X 0,Y 279.788,Z 304.454,A -85,B 0,C 180,E1 -18503.496,E2 -18503.496} C_VEL
LIN {X 0,Y 280.931,Z 307.381,A -85,B 0,C 180,E1 -18505.646,E2 -18505.646} C_VEL
LIN {X 0,Y 282.073,Z 311.553,A -85,B 0,C 180,E1 -18507.902,E2 -18507.902} C_VEL
LIN {X 0,Y 283.071,Z 317.18,A -85,B 0,C 180,E1 -18510.34,E2 -18510.34} C_VEL
LIN {X 0,Y 283.433,Z 323.638,A -85,B 0,C 180,E1 -18512.695,E2 -18512.695} C_VEL
LIN {X 0,Y 280.472,Z 329.866,A -85,B 0,C 180,E1 -18513.991,E2 -18513.991} C_VEL
LIN {X 0,Y 276.001,Z 338.037,A -85,B 0,C 180,E1 -18515.957,E2 -18515.957} C_VEL
LIN {X 0,Y 271.444,Z 345.846,A -85,B 0,C 180,E1 -18518.349,E2 -18518.349} C_VEL
LIN {X 0,Y 267.415,Z 352.122,A -85,B 0,C 180,E1 -18520.821,E2 -18520.821} C_VEL
LIN {X 0,Y 263.429,Z 357.623,A -85,B 0,C 180,E1 -18523.732,E2 -18523.732} C_VEL
LIN {X 0,Y 260.969,Z 360.672,A -85,B 0,C 180,E1 -18525.973,E2 -18525.973} C_VEL
LIN {X 0,Y 258.181,Z 363.445,A -85,B 0,C 180,E1 -18529.015,E2 -18529.015} C_VEL
LIN {X 0,Y 256.612,Z 364.625,A -85,B 0,C 180,E1 -18532.129,E2 -18532.129} C_VEL
LIN {X 0,Y 255.421,Z 364.4,A -85,B 0,C 180,E1 -18535.265,E2 -18535.265} C_VEL
LIN {X 0,Y 254.85,Z 363.739,A -85,B 0,C 180,E1 -18536.838,E2 -18536.838} C_VEL
LIN {X 0,Y 254.308,Z 361.193,A -85,B 0,C 180,E1 -18540,E2 -18540} C_VEL
LIN {X 0,Y 254.283,Z 358.249,A -85,B 0,C 180,E1 -18542.376,E2 -18542.376} C_VEL
LIN {X 0,Y 254.307,Z 353.364,A -85,B 0,C 180,E1 -18545.252,E2 -18545.252} C_VEL
LIN {X 0,Y 254.666,Z 347.362,A -85,B 0,C 180,E1 -18547.931,E2 -18547.931} C_VEL
LIN {X 0,Y 255.224,Z 339.37,A -85,B 0,C 180,E1 -18550.712,E2 -18550.712} C_VEL
LIN {X 0,Y 255.96,Z 330.875,A -85,B 0,C 180,E1 -18553.093,E2 -18553.093} C_VEL
LIN {X 0,Y 256.86,Z 322.3,A -85,B 0,C 180,E1 -18555.066,E2 -18555.066} C_VEL
LIN {X 0,Y 257.813,Z 311.965,A -85,B 0,C 180,E1 -18557.041,E2 -18557.041} C_VEL
LIN {X 0,Y 258.972,Z 300.895,A -85,B 0,C 180,E1 -18558.78,E2 -18558.78} C_VEL
LIN {X 0,Y 260.007,Z 290.115,A -85,B 0,C 180,E1 -18560.16,E2 -18560.16} C_VEL
LIN {X 0,Y 257.875,Z 277.614,A -85,B 0,C 180,E1 -18561.533,E2 -18561.533} C_VEL
LIN {X 0,Y 255.492,Z 264.012,A -85,B 0,C 180,E1 -18562.716,E2 -18562.716} C_VEL
LIN {X 0,Y 254.595,Z 258.158,A -85,B 0,C 180,E1 -18563.164,E2 -18563.164} C_VEL
LIN {X 0,Y 254.668,Z 256.764,A -85,B 0,C 180,E1 -18564.889,E2 -18564.889} C_VEL
LIN {X 0,Y 255.044,Z 256.718,A -85,B 0,C 180,E1 -18568.139,E2 -18568.139} C_VEL
LIN {X 0,Y 255.441,Z 256.667,A -85,B 0,C 180,E1 -18571.517,E2 -18571.517} C_VEL
LIN {X 0,Y 255.827,Z 256.617,A -85,B 0,C 180,E1 -18575.234,E2 -18575.234} C_VEL
LIN {X 0,Y 256.011,Z 256.597,A -85,B 0,C 180,E1 -18577.239,E2 -18577.239} C_VEL
LIN {X 0,Y 256.056,Z 256.59,A -85,B 0,C 180,E1 -18581.204,E2 -18581.204} C_VEL
LIN {X 0,Y 256.043,Z 256.59,A -85,B 0,C 180,E1 -18585.534,E2 -18585.534} C_VEL
LIN {X 0,Y 256.043,Z 256.592,A -85,B 0,C 180,E1 -18588.794,E2 -18588.794} C_VEL
LIN {X 0,Y 256.128,Z 256.581,A -85,B 0,C 180,E1 -18592.867,E2 -18592.867} C_VEL
LIN {X 0,Y 256.069,Z 256.59,A -85,B 0,C 180,E1 -18596.707,E2 -18596.707} C_VEL
LIN {X 0,Y 256.061,Z 256.59,A -85,B 0,C 180,E1 -18600.393,E2 -18600.393} C_VEL
LIN {X 0,Y 256.165,Z 256.576,A -85,B 0,C 180,E1 -18604.874,E2 -18604.874} C_VEL
LIN {X 0,Y 256.166,Z 256.574,A -85,B 0,C 180,E1 -18609.104,E2 -18609.104} C_VEL
LIN {X 0,Y 256.304,Z 256.558,A -85,B 0,C 180,E1 -18614.085,E2 -18614.085} C_VEL
LIN {X 0,Y 256.299,Z 256.558,A -85,B 0,C 180,E1 -18618.933,E2 -18618.933} C_VEL
LIN {X 0,Y 256.492,Z 256.538,A -85,B 0,C 180,E1 -18622.125,E2 -18622.125} C_VEL
LIN {X 0,Y 256.446,Z 256.539,A -85,B 0,C 180,E1 -18626.858,E2 -18626.858} C_VEL
LIN {X 0,Y 256.699,Z 256.51,A -85,B 0,C 180,E1 -18628.431,E2 -18628.431} C_VEL
LIN {X 0,Y 256.664,Z 256.699,A -85,B 0,C 180,E1 -18631.961,E2 -18631.961} C_VEL
LIN {X 0,Y 256.8,Z 262.354,A -85,B 0,C 180,E1 -18635.496,E2 -18635.496} C_VEL
LIN {X 0,Y 256.422,Z 268.853,A -85,B 0,C 180,E1 -18639.465,E2 -18639.465} C_VEL
LIN {X 0,Y 256.059,Z 275.432,A -85,B 0,C 180,E1 -18643.491,E2 -18643.491} C_VEL
LIN {X 0,Y 255.835,Z 280.685,A -85,B 0,C 180,E1 -18646.691,E2 -18646.691} C_VEL
LIN {X 0,Y 257.816,Z 291.348,A -85,B 0,C 180,E1 -18647.449,E2 -18647.449} C_VEL
LIN {X 0,Y 259.381,Z 301.097,A -85,B 0,C 180,E1 -18648.359,E2 -18648.359} C_VEL
LIN {X 0,Y 260.38,Z 308.6,A -85,B 0,C 180,E1 -18649.23,E2 -18649.23} C_VEL
LIN {X 0,Y 259.661,Z 317.474,A -85,B 0,C 180,E1 -18650.373,E2 -18650.373} C_VEL
LIN {X 0,Y 258.575,Z 326.816,A -85,B 0,C 180,E1 -18651.908,E2 -18651.908} C_VEL
LIN {X 0,Y 257.721,Z 333.613,A -85,B 0,C 180,E1 -18653.292,E2 -18653.292} C_VEL
LIN {X 0,Y 256.832,Z 340.404,A -85,B 0,C 180,E1 -18654.979,E2 -18654.979} C_VEL
LIN {X 0,Y 256.14,Z 345.406,A -85,B 0,C 180,E1 -18656.479,E2 -18656.479} C_VEL
LIN {X 0,Y 255.468,Z 350.418,A -85,B 0,C 180,E1 -18658.317,E2 -18658.317} C_VEL
LIN {X 0,Y 254.869,Z 355.016,A -85,B 0,C 180,E1 -18660.463,E2 -18660.463} C_VEL
LIN {X 0,Y 254.41,Z 358.432,A -85,B 0,C 180,E1 -18662.594,E2 -18662.594} C_VEL
LIN {X 0,Y 254.074,Z 361.384,A -85,B 0,C 180,E1 -18665.513,E2 -18665.513} C_VEL
LIN {X 0,Y 254.063,Z 362.394,A -85,B 0,C 180,E1 -18667.486,E2 -18667.486} C_VEL
LIN {X 0,Y 254.251,Z 362.62,A -85,B 0,C 180,E1 -18669.477,E2 -18669.477} C_VEL
LIN {X 0,Y 254.694,Z 361.849,A -85,B 0,C 180,E1 -18671.837,E2 -18671.837} C_VEL
LIN {X 0,Y 255.468,Z 359.837,A -85,B 0,C 180,E1 -18674.334,E2 -18674.334} C_VEL
LIN {X 0,Y 256.435,Z 356.588,A -85,B 0,C 180,E1 -18676.751,E2 -18676.751} C_VEL
LIN {X 0,Y 257.282,Z 353.58,A -85,B 0,C 180,E1 -18678.377,E2 -18678.377} C_VEL
LIN {X 0,Y 258.695,Z 348.319,A -85,B 0,C 180,E1 -18680.55,E2 -18680.55} C_VEL
LIN {X 0,Y 259.961,Z 343.105,A -85,B 0,C 180,E1 -18682.257,E2 -18682.257} C_VEL
LIN {X 0,Y 261.363,Z 337.409,A -85,B 0,C 180,E1 -18683.774,E2 -18683.774} C_VEL
LIN {X 0,Y 262.869,Z 330.428,A -85,B 0,C 180,E1 -18685.298,E2 -18685.298} C_VEL
LIN {X 0,Y 264.162,Z 323.46,A -85,B 0,C 180,E1 -18686.552,E2 -18686.552} C_VEL
LIN {X 0,Y 265.286,Z 316.733,A -85,B 0,C 180,E1 -18687.556,E2 -18687.556} C_VEL
LIN {X 0,Y 264.468,Z 308.567,A -85,B 0,C 180,E1 -18688.788,E2 -18688.788} C_VEL
LIN {X 0,Y 262.906,Z 300.168,A -85,B 0,C 180,E1 -18689.919,E2 -18689.919} C_VEL
LIN {X 0,Y 260.443,Z 290.769,A -85,B 0,C 180,E1 -18691.056,E2 -18691.056} C_VEL
LIN {X 0,Y 257.639,Z 282.393,A -85,B 0,C 180,E1 -18691.964,E2 -18691.964} C_VEL
LIN {X 0,Y 258.19,Z 276.281,A -85,B 0,C 180,E1 -18695.901,E2 -18695.901} C_VEL
LIN {X 0,Y 258.682,Z 271.025,A -85,B 0,C 180,E1 -18699.317,E2 -18699.317} C_VEL
LIN {X 0,Y 258.346,Z 266.864,A -85,B 0,C 180,E1 -18702.201,E2 -18702.201} C_VEL
LIN {X 0,Y 257.557,Z 261.989,A -85,B 0,C 180,E1 -18705.783,E2 -18705.783} C_VEL
LIN {X 0,Y 256.364,Z 256.554,A -85,B 0,C 180,E1 -18710.034,E2 -18710.034} C_VEL
LIN {X 0,Y 256.506,Z 256.536,A -85,B 0,C 180,E1 -18712.126,E2 -18712.126} C_VEL
LIN {X 0,Y 256.497,Z 256.536,A -85,B 0,C 180,E1 -18716.858,E2 -18716.858} C_VEL
LIN {X 0,Y 256.767,Z 256.501,A -85,B 0,C 180,E1 -18720,E2 -18720} C_VEL
LIN {X 0,Y 256.497,Z 256.535,A -85,B 0,C 180,E1 -18723.141,E2 -18723.141} C_VEL
LIN {X 0,Y 256.497,Z 256.534,A -85,B 0,C 180,E1 -18727.874,E2 -18727.874} C_VEL
LIN {X 0,Y 256.296,Z 256.56,A -85,B 0,C 180,E1 -18732.672,E2 -18732.672} C_VEL
LIN {X 0,Y 256.284,Z 256.557,A -85,B 0,C 180,E1 -18736.302,E2 -18736.302} C_VEL
LIN {X 0,Y 256.155,Z 256.574,A -85,B 0,C 180,E1 -18741.117,E2 -18741.117} C_VEL
LIN {X 0,Y 256.085,Z 256.585,A -85,B 0,C 180,E1 -18742.317,E2 -18742.317} C_VEL
LIN {X 0,Y 255.428,Z 256.673,A -85,B 0,C 180,E1 -18743.63,E2 -18743.63} C_VEL
LIN {X 0,Y 252.624,Z 257.024,A -85,B 0,C 180,E1 -18745.774,E2 -18745.774} C_VEL
LIN {X 0,Y 250.224,Z 257.317,A -85,B 0,C 180,E1 -18747.517,E2 -18747.517} C_VEL
LIN {X 0,Y 249.165,Z 257.446,A -85,B 0,C 180,E1 -18748.868,E2 -18748.868} C_VEL
LIN {X 0,Y 249.063,Z 257.456,A -85,B 0,C 180,E1 -18749.326,E2 -18749.326} C_VEL
LIN {X 0,Y 249.034,Z 257.46,A -85,B 0,C 180,E1 -18752.425,E2 -18752.425} C_VEL
LIN {X 0,Y 249.064,Z 257.46,A -85,B 0,C 180,E1 -18756.34,E2 -18756.34} C_VEL
LIN {X 0,Y 249.026,Z 257.465,A -85,B 0,C 180,E1 -18760.474,E2 -18760.474} C_VEL
LIN {X 0,Y 249.212,Z 257.526,A -85,B 0,C 180,E1 -18764.278,E2 -18764.278} C_VEL
LIN {X 0,Y 250.252,Z 263.302,A -85,B 0,C 180,E1 -18769.311,E2 -18769.311} C_VEL
LIN {X 0,Y 250.826,Z 266.44,A -85,B 0,C 180,E1 -18771.944,E2 -18771.944} C_VEL
LIN {X 0,Y 250.79,Z 269.42,A -85,B 0,C 180,E1 -18774.359,E2 -18774.359} C_VEL
LIN {X 0,Y 249.984,Z 273.376,A -85,B 0,C 180,E1 -18777.338,E2 -18777.338} C_VEL
LIN {X 0,Y 250.592,Z 283.639,A -85,B 0,C 180,E1 -18780.391,E2 -18780.391} C_VEL
LIN {X 0,Y 251.396,Z 295.245,A -85,B 0,C 180,E1 -18783.456,E2 -18783.456} C_VEL
LIN {X 0,Y 251.543,Z 298.426,A -85,B 0,C 180,E1 -18784.188,E2 -18784.188} C_VEL
LIN {X 0,Y 254.468,Z 309.548,A -85,B 0,C 180,E1 -18785.124,E2 -18785.124} C_VEL
LIN {X 0,Y 255.182,Z 322.193,A -85,B 0,C 180,E1 -18786.184,E2 -18786.184} C_VEL
LIN {X 0,Y 255.51,Z 331.191,A -85,B 0,C 180,E1 -18787.183,E2 -18787.183} C_VEL
LIN {X 0,Y 255.545,Z 338.909,A -85,B 0,C 180,E1 -18788.206,E2 -18788.206} C_VEL
LIN {X 0,Y 254.349,Z 346.939,A -85,B 0,C 180,E1 -18789.372,E2 -18789.372} C_VEL
LIN {X 0,Y 253.123,Z 353.638,A -85,B 0,C 180,E1 -18790.538,E2 -18790.538} C_VEL
LIN {X 0,Y 251.944,Z 359.523,A -85,B 0,C 180,E1 -18791.749,E2 -18791.749} C_VEL
LIN {X 0,Y 250.86,Z 365.77,A -85,B 0,C 180,E1 -18793.312,E2 -18793.312} C_VEL
LIN {X 0,Y 249.811,Z 371.132,A -85,B 0,C 180,E1 -18794.916,E2 -18794.916} C_VEL
LIN {X 0,Y 248.61,Z 376.611,A -85,B 0,C 180,E1 -18796.929,E2 -18796.929} C_VEL
LIN {X 0,Y 247.773,Z 381.754,A -85,B 0,C 180,E1 -18799.376,E2 -18799.376} C_VEL
LIN {X 0,Y 247.285,Z 385.523,A -85,B 0,C 180,E1 -18801.831,E2 -18801.831} C_VEL
LIN {X 0,Y 247.163,Z 387.261,A -85,B 0,C 180,E1 -18803.469,E2 -18803.469} C_VEL
LIN {X 0,Y 247.059,Z 388.473,A -85,B 0,C 180,E1 -18805.105,E2 -18805.105} C_VEL
LIN {X 0,Y 247.14,Z 389.208,A -85,B 0,C 180,E1 -18806.74,E2 -18806.74} C_VEL
LIN {X 0,Y 247.213,Z 389.462,A -85,B 0,C 180,E1 -18808.371,E2 -18808.371} C_VEL
LIN {X 0,Y 247.336,Z 389.199,A -85,B 0,C 180,E1 -18810,E2 -18810} C_VEL
LIN {X 0,Y 247.321,Z 387.929,A -85,B 0,C 180,E1 -18812.24,E2 -18812.24} C_VEL
LIN {X 0,Y 247.022,Z 389.122,A -85,B 0,C 180,E1 -18815.264,E2 -18815.264} C_VEL
LIN {X 0,Y 247.236,Z 389.064,A -85,B 0,C 180,E1 -18818.171,E2 -18818.171} C_VEL
LIN {X 0,Y 248.124,Z 387.614,A -85,B 0,C 180,E1 -18821.436,E2 -18821.436} C_VEL
LIN {X 0,Y 249.831,Z 384.759,A -85,B 0,C 180,E1 -18824.666,E2 -18824.666} C_VEL
LIN {X 0,Y 252.695,Z 380.388,A -85,B 0,C 180,E1 -18827.815,E2 -18827.815} C_VEL
LIN {X 0,Y 255.143,Z 376.147,A -85,B 0,C 180,E1 -18830.14,E2 -18830.14} C_VEL
LIN {X 0,Y 258.189,Z 370.994,A -85,B 0,C 180,E1 -18832.401,E2 -18832.401} C_VEL
LIN {X 0,Y 262.628,Z 363.635,A -85,B 0,C 180,E1 -18834.928,E2 -18834.928} C_VEL
LIN {X 0,Y 267.733,Z 354.74,A -85,B 0,C 180,E1 -18837.347,E2 -18837.347} C_VEL
LIN {X 0,Y 270.488,Z 349.036,A -85,B 0,C 180,E1 -18838.73,E2 -18838.73} C_VEL
LIN {X 0,Y 272.495,Z 341.996,A -85,B 0,C 180,E1 -18840.582,E2 -18840.582} C_VEL
LIN {X 0,Y 273.949,Z 333.082,A -85,B 0,C 180,E1 -18843.083,E2 -18843.083} C_VEL
LIN {X 0,Y 274.549,Z 325.326,A -85,B 0,C 180,E1 -18845.508,E2 -18845.508} C_VEL
LIN {X 0,Y 274.76,Z 319.593,A -85,B 0,C 180,E1 -18847.539,E2 -18847.539} C_VEL
LIN {X 0,Y 274.765,Z 315.828,A -85,B 0,C 180,E1 -18849.124,E2 -18849.124} C_VEL
LIN {X 0,Y 274.551,Z 312.924,A -85,B 0,C 180,E1 -18850.673,E2 -18850.673} C_VEL
LIN {X 0,Y 274.23,Z 311.202,A -85,B 0,C 180,E1 -18851.994,E2 -18851.994} C_VEL
LIN {X 0,Y 273.806,Z 309.368,A -85,B 0,C 180,E1 -18854.053,E2 -18854.053} C_VEL
LIN {X 0,Y 273.746,Z 308.187,A -85,B 0,C 180,E1 -18856.117,E2 -18856.117} C_VEL
LIN {X 0,Y 273.993,Z 307.768,A -85,B 0,C 180,E1 -18858.171,E2 -18858.171} C_VEL
LIN {X 0,Y 274.583,Z 308.021,A -85,B 0,C 180,E1 -18860.217,E2 -18860.217} C_VEL
LIN {X 0,Y 275.33,Z 309.29,A -85,B 0,C 180,E1 -18862.308,E2 -18862.308} C_VEL
LIN {X 0,Y 276.471,Z 312.469,A -85,B 0,C 180,E1 -18865.142,E2 -18865.142} C_VEL
LIN {X 0,Y 277.434,Z 317.159,A -85,B 0,C 180,E1 -18867.861,E2 -18867.861} C_VEL
LIN {X 0,Y 278,Z 322.786,A -85,B 0,C 180,E1 -18870.404,E2 -18870.404} C_VEL
LIN {X 0,Y 277.824,Z 327.241,A -85,B 0,C 180,E1 -18872.096,E2 -18872.096} C_VEL
LIN {X 0,Y 272.147,Z 337.179,A -85,B 0,C 180,E1 -18874.37,E2 -18874.37} C_VEL
LIN {X 0,Y 267.132,Z 345.194,A -85,B 0,C 180,E1 -18876.757,E2 -18876.757} C_VEL
LIN {X 0,Y 263.265,Z 350.832,A -85,B 0,C 180,E1 -18878.876,E2 -18878.876} C_VEL
LIN {X 0,Y 258.778,Z 356.787,A -85,B 0,C 180,E1 -18881.801,E2 -18881.801} C_VEL
LIN {X 0,Y 255.844,Z 360.165,A -85,B 0,C 180,E1 -18884.056,E2 -18884.056} C_VEL
LIN {X 0,Y 252.731,Z 363.301,A -85,B 0,C 180,E1 -18887.146,E2 -18887.146} C_VEL
LIN {X 0,Y 251.27,Z 364.33,A -85,B 0,C 180,E1 -18888.709,E2 -18888.709} C_VEL
LIN {X 0,Y 249.604,Z 365.252,A -85,B 0,C 180,E1 -18891.907,E2 -18891.907} C_VEL
LIN {X 0,Y 248.354,Z 364.729,A -85,B 0,C 180,E1 -18895.13,E2 -18895.13} C_VEL
LIN {X 0,Y 247.401,Z 362.709,A -85,B 0,C 180,E1 -18898.372,E2 -18898.372} C_VEL
LIN {X 0,Y 247.183,Z 360.17,A -85,B 0,C 180,E1 -18900.815,E2 -18900.815} C_VEL
LIN {X 0,Y 247.205,Z 356.694,A -85,B 0,C 180,E1 -18903.26,E2 -18903.26} C_VEL
LIN {X 0,Y 247.333,Z 351.606,A -85,B 0,C 180,E1 -18905.989,E2 -18905.989} C_VEL
LIN {X 0,Y 247.676,Z 345.478,A -85,B 0,C 180,E1 -18908.568,E2 -18908.568} C_VEL
LIN {X 0,Y 248.221,Z 338.251,A -85,B 0,C 180,E1 -18911.018,E2 -18911.018} C_VEL
LIN {X 0,Y 249.021,Z 329.385,A -85,B 0,C 180,E1 -18913.464,E2 -18913.464} C_VEL
LIN {X 0,Y 249.94,Z 320.49,A -85,B 0,C 180,E1 -18915.494,E2 -18915.494} C_VEL
LIN {X 0,Y 250.969,Z 309.809,A -85,B 0,C 180,E1 -18917.508,E2 -18917.508} C_VEL
LIN {X 0,Y 252.203,Z 298.105,A -85,B 0,C 180,E1 -18919.303,E2 -18919.303} C_VEL
LIN {X 0,Y 252.828,Z 290.063,A -85,B 0,C 180,E1 -18920.333,E2 -18920.333} C_VEL
LIN {X 0,Y 250.509,Z 276.474,A -85,B 0,C 180,E1 -18921.853,E2 -18921.853} C_VEL
LIN {X 0,Y 247.932,Z 261.521,A -85,B 0,C 180,E1 -18923.134,E2 -18923.134} C_VEL
LIN {X 0,Y 247.529,Z 258.572,A -85,B 0,C 180,E1 -18923.341,E2 -18923.341} C_VEL
LIN {X 0,Y 247.574,Z 257.647,A -85,B 0,C 180,E1 -18924.714,E2 -18924.714} C_VEL
LIN {X 0,Y 248.064,Z 257.584,A -85,B 0,C 180,E1 -18928.793,E2 -18928.793} C_VEL
LIN {X 0,Y 248.482,Z 257.531,A -85,B 0,C 180,E1 -18932.507,E2 -18932.507} C_VEL
LIN {X 0,Y 248.789,Z 257.492,A -85,B 0,C 180,E1 -18934.993,E2 -18934.993} C_VEL
LIN {X 0,Y 248.983,Z 257.469,A -85,B 0,C 180,E1 -18938.389,E2 -18938.389} C_VEL
LIN {X 0,Y 249.004,Z 257.467,A -85,B 0,C 180,E1 -18942.79,E2 -18942.79} C_VEL
LIN {X 0,Y 249.005,Z 257.467,A -85,B 0,C 180,E1 -18947.36,E2 -18947.36} C_VEL
LIN {X 0,Y 249.043,Z 257.462,A -85,B 0,C 180,E1 -18952.201,E2 -18952.201} C_VEL
LIN {X 0,Y 249.046,Z 257.462,A -85,B 0,C 180,E1 -18955.639,E2 -18955.639} C_VEL
LIN {X 0,Y 249.006,Z 257.465,A -85,B 0,C 180,E1 -18959.466,E2 -18959.466} C_VEL
LIN {X 0,Y 249.046,Z 257.461,A -85,B 0,C 180,E1 -18963.159,E2 -18963.159} C_VEL
LIN {X 0,Y 249.061,Z 257.459,A -85,B 0,C 180,E1 -18966.73,E2 -18966.73} C_VEL
LIN {X 0,Y 249.113,Z 257.456,A -85,B 0,C 180,E1 -18970.211,E2 -18970.211} C_VEL
LIN {X 0,Y 249.245,Z 257.434,A -85,B 0,C 180,E1 -18973.622,E2 -18973.622} C_VEL
LIN {X 0,Y 249.247,Z 257.438,A -85,B 0,C 180,E1 -18978.616,E2 -18978.616} C_VEL
LIN {X 0,Y 249.437,Z 257.417,A -85,B 0,C 180,E1 -18981.901,E2 -18981.901} C_VEL
LIN {X 0,Y 249.257,Z 257.436,A -85,B 0,C 180,E1 -18985.147,E2 -18985.147} C_VEL
LIN {X 0,Y 249.66,Z 257.387,A -85,B 0,C 180,E1 -18988.387,E2 -18988.387} C_VEL
LIN {X 0,Y 249.669,Z 257.578,A -85,B 0,C 180,E1 -18991.613,E2 -18991.613} C_VEL
LIN {X 0,Y 249.843,Z 262.593,A -85,B 0,C 180,E1 -18994.841,E2 -18994.841} C_VEL
LIN {X 0,Y 249.444,Z 269.434,A -85,B 0,C 180,E1 -18999.109,E2 -18999.109} C_VEL
LIN {X 0,Y 249.066,Z 275.821,A -85,B 0,C 180,E1 -19003.046,E2 -19003.046} C_VEL
LIN {X 0,Y 248.861,Z 281.126,A -85,B 0,C 180,E1 -19006.261,E2 -19006.261} C_VEL
LIN {X 0,Y 250.675,Z 290.888,A -85,B 0,C 180,E1 -19006.963,E2 -19006.963} C_VEL
LIN {X 0,Y 252.199,Z 300.301,A -85,B 0,C 180,E1 -19007.85,E2 -19007.85} C_VEL
LIN {X 0,Y 253.454,Z 310.163,A -85,B 0,C 180,E1 -19009.014,E2 -19009.014} C_VEL
LIN {X 0,Y 252.528,Z 319.855,A -85,B 0,C 180,E1 -19010.358,E2 -19010.358} C_VEL
LIN {X 0,Y 251.426,Z 328.468,A -85,B 0,C 180,E1 -19011.88,E2 -19011.88} C_VEL
LIN {X 0,Y 250.7,Z 334.247,A -85,B 0,C 180,E1 -19013.108,E2 -19013.108} C_VEL
LIN {X 0,Y 249.974,Z 339.804,A -85,B 0,C 180,E1 -19014.5,E2 -19014.5} C_VEL
LIN {X 0,Y 249.165,Z 345.368,A -85,B 0,C 180,E1 -19016.176,E2 -19016.176} C_VEL
LIN {X 0,Y 248.417,Z 350.772,A -85,B 0,C 180,E1 -19018.198,E2 -19018.198} C_VEL
LIN {X 0,Y 247.968,Z 354.122,A -85,B 0,C 180,E1 -19019.735,E2 -19019.735} C_VEL
LIN {X 0,Y 247.525,Z 357.363,A -85,B 0,C 180,E1 -19021.592,E2 -19021.592} C_VEL
LIN {X 0,Y 247.299,Z 358.926,A -85,B 0,C 180,E1 -19022.681,E2 -19022.681} C_VEL
LIN {X 0,Y 247.031,Z 361.086,A -85,B 0,C 180,E1 -19024.68,E2 -19024.68} C_VEL
LIN {X 0,Y 246.963,Z 362.676,A -85,B 0,C 180,E1 -19027.172,E2 -19027.172} C_VEL
LIN {X 0,Y 247.218,Z 362.99,A -85,B 0,C 180,E1 -19029.864,E2 -19029.864} C_VEL
LIN {X 0,Y 247.788,Z 362.05,A -85,B 0,C 180,E1 -19032.486,E2 -19032.486} C_VEL
LIN {X 0,Y 248.621,Z 359.908,A -85,B 0,C 180,E1 -19035.033,E2 -19035.033} C_VEL
LIN {X 0,Y 249.693,Z 356.418,A -85,B 0,C 180,E1 -19037.505,E2 -19037.505} C_VEL
LIN {X 0,Y 251.174,Z 351.528,A -85,B 0,C 180,E1 -19039.942,E2 -19039.942} C_VEL
LIN {X 0,Y 252.861,Z 345.253,A -85,B 0,C 180,E1 -19042.304,E2 -19042.304} C_VEL
LIN {X 0,Y 254.742,Z 337.966,A -85,B 0,C 180,E1 -19044.342,E2 -19044.342} C_VEL
LIN {X 0,Y 256.43,Z 330.541,A -85,B 0,C 180,E1 -19045.995,E2 -19045.995} C_VEL
LIN {X 0,Y 257.933,Z 323.045,A -85,B 0,C 180,E1 -19047.349,E2 -19047.349} C_VEL
LIN {X 0,Y 258.727,Z 317.291,A -85,B 0,C 180,E1 -19048.243,E2 -19048.243} C_VEL
LIN {X 0,Y 257.927,Z 309.347,A -85,B 0,C 180,E1 -19049.503,E2 -19049.503} C_VEL
LIN {X 0,Y 256.426,Z 301.064,A -85,B 0,C 180,E1 -19050.677,E2 -19050.677} C_VEL
LIN {X 0,Y 253.814,Z 291.363,A -85,B 0,C 180,E1 -19051.918,E2 -19051.918} C_VEL
LIN {X 0,Y 250.901,Z 282.737,A -85,B 0,C 180,E1 -19052.923,E2 -19052.923} C_VEL
LIN {X 0,Y 251.534,Z 276.235,A -85,B 0,C 180,E1 -19057.226,E2 -19057.226} C_VEL
LIN {X 0,Y 251.857,Z 272.706,A -85,B 0,C 180,E1 -19059.585,E2 -19059.585} C_VEL
LIN {X 0,Y 251.607,Z 269.194,A -85,B 0,C 180,E1 -19062.106,E2 -19062.106} C_VEL
LIN {X 0,Y 250.902,Z 264.74,A -85,B 0,C 180,E1 -19065.398,E2 -19065.398} C_VEL
LIN {X 0,Y 249.612,Z 258.651,A -85,B 0,C 180,E1 -19070.274,E2 -19070.274} C_VEL
LIN {X 0,Y 249.414,Z 257.419,A -85,B 0,C 180,E1 -19071.421,E2 -19071.421} C_VEL
LIN {X 0,Y 249.442,Z 257.415,A -85,B 0,C 180,E1 -19073.529,E2 -19073.529} C_VEL
LIN {X 0,Y 249.677,Z 257.386,A -85,B 0,C 180,E1 -19078.387,E2 -19078.387} C_VEL
LIN {X 0,Y 249.677,Z 257.383,A -85,B 0,C 180,E1 -19081.613,E2 -19081.613} C_VEL
LIN {X 0,Y 249.438,Z 257.412,A -85,B 0,C 180,E1 -19086.471,E2 -19086.471} C_VEL
LIN {X 0,Y 249.345,Z 257.427,A -85,B 0,C 180,E1 -19089.736,E2 -19089.736} C_VEL
LIN {X 0,Y 249.207,Z 257.444,A -85,B 0,C 180,E1 -19094.703,E2 -19094.703} C_VEL
LIN {X 0,Y 249.141,Z 257.449,A -85,B 0,C 180,E1 -19098.077,E2 -19098.077} C_VEL
LIN {X 0,Y 249.046,Z 257.457,A -85,B 0,C 180,E1 -19102.31,E2 -19102.31} C_VEL
LIN {X 0,Y 249.118,Z 257.455,A -85,B 0,C 180,E1 -19105.476,E2 -19105.476} C_VEL
LIN {X 0,Y 249.063,Z 257.456,A -85,B 0,C 180,E1 -19109.326,E2 -19109.326} C_VEL
LIN {X 0,Y 248.355,Z 257.549,A -85,B 0,C 180,E1 -19110.675,E2 -19110.675} C_VEL
LIN {X 0,Y 245.504,Z 257.902,A -85,B 0,C 180,E1 -19112.875,E2 -19112.875} C_VEL
LIN {X 0,Y 243.103,Z 258.2,A -85,B 0,C 180,E1 -19114.666,E2 -19114.666} C_VEL
LIN {X 0,Y 242.067,Z 258.332,A -85,B 0,C 180,E1 -19116.055,E2 -19116.055} C_VEL
LIN {X 0,Y 241.978,Z 258.336,A -85,B 0,C 180,E1 -19116.526,E2 -19116.526} C_VEL
LIN {X 0,Y 241.969,Z 258.34,A -85,B 0,C 180,E1 -19119.717,E2 -19119.717} C_VEL
LIN {X 0,Y 242.188,Z 258.523,A -85,B 0,C 180,E1 -19124.433,E2 -19124.433} C_VEL
LIN {X 0,Y 243.049,Z 263.328,A -85,B 0,C 180,E1 -19128.748,E2 -19128.748} C_VEL
LIN {X 0,Y 243.589,Z 266.104,A -85,B 0,C 180,E1 -19131.169,E2 -19131.169} C_VEL
LIN {X 0,Y 243.797,Z 269.251,A -85,B 0,C 180,E1 -19133.82,E2 -19133.82} C_VEL
LIN {X 0,Y 243.497,Z 271.051,A -85,B 0,C 180,E1 -19135.122,E2 -19135.122} C_VEL
LIN {X 0,Y 243.966,Z 280.595,A -85,B 0,C 180,E1 -19138.282,E2 -19138.282} C_VEL
LIN {X 0,Y 244.525,Z 290.567,A -85,B 0,C 180,E1 -19141.222,E2 -19141.222} C_VEL
LIN {X 0,Y 244.929,Z 298.127,A -85,B 0,C 180,E1 -19143.192,E2 -19143.192} C_VEL
LIN {X 0,Y 248.384,Z 311.202,A -85,B 0,C 180,E1 -19144.377,E2 -19144.377} C_VEL
LIN {X 0,Y 248.884,Z 322.049,A -85,B 0,C 180,E1 -19145.354,E2 -19145.354} C_VEL
LIN {X 0,Y 249.048,Z 330.594,A -85,B 0,C 180,E1 -19146.325,E2 -19146.325} C_VEL
LIN {X 0,Y 249.01,Z 339.754,A -85,B 0,C 180,E1 -19147.603,E2 -19147.603} C_VEL
LIN {X 0,Y 247.76,Z 347.538,A -85,B 0,C 180,E1 -19148.797,E2 -19148.797} C_VEL
LIN {X 0,Y 246.466,Z 354.071,A -85,B 0,C 180,E1 -19149.99,E2 -19149.99} C_VEL
LIN {X 0,Y 245.181,Z 359.823,A -85,B 0,C 180,E1 -19151.227,E2 -19151.227} C_VEL
LIN {X 0,Y 244.074,Z 365.954,A -85,B 0,C 180,E1 -19152.834,E2 -19152.834} C_VEL
LIN {X 0,Y 242.702,Z 372.392,A -85,B 0,C 180,E1 -19154.894,E2 -19154.894} C_VEL
LIN {X 0,Y 241.668,Z 376.602,A -85,B 0,C 180,E1 -19156.547,E2 -19156.547} C_VEL
LIN {X 0,Y 241.053,Z 380.107,A -85,B 0,C 180,E1 -19158.224,E2 -19158.224} C_VEL
LIN {X 0,Y 240.37,Z 384.178,A -85,B 0,C 180,E1 -19160.746,E2 -19160.746} C_VEL
LIN {X 0,Y 240.074,Z 387.019,A -85,B 0,C 180,E1 -19163.276,E2 -19163.276} C_VEL
LIN {X 0,Y 239.969,Z 388.173,A -85,B 0,C 180,E1 -19164.96,E2 -19164.96} C_VEL
LIN {X 0,Y 240.047,Z 388.847,A -85,B 0,C 180,E1 -19166.643,E2 -19166.643} C_VEL
LIN {X 0,Y 240.133,Z 389.042,A -85,B 0,C 180,E1 -19168.323,E2 -19168.323} C_VEL
LIN {X 0,Y 240.25,Z 388.747,A -85,B 0,C 180,E1 -19170,E2 -19170} C_VEL
LIN {X 0,Y 240.214,Z 387.239,A -85,B 0,C 180,E1 -19172.62,E2 -19172.62} C_VEL
LIN {X 0,Y 239.984,Z 388.424,A -85,B 0,C 180,E1 -19175.315,E2 -19175.315} C_VEL
LIN {X 0,Y 240.188,Z 388.623,A -85,B 0,C 180,E1 -19178.413,E2 -19178.413} C_VEL
LIN {X 0,Y 241.151,Z 387.446,A -85,B 0,C 180,E1 -19181.772,E2 -19181.772} C_VEL
LIN {X 0,Y 242.977,Z 384.841,A -85,B 0,C 180,E1 -19185.089,E2 -19185.089} C_VEL
LIN {X 0,Y 245.966,Z 380.829,A -85,B 0,C 180,E1 -19188.319,E2 -19188.319} C_VEL
LIN {X 0,Y 248.519,Z 376.848,A -85,B 0,C 180,E1 -19190.702,E2 -19190.702} C_VEL
LIN {X 0,Y 251.708,Z 371.997,A -85,B 0,C 180,E1 -19193.011,E2 -19193.011} C_VEL
LIN {X 0,Y 257.045,Z 364.007,A -85,B 0,C 180,E1 -19195.943,E2 -19195.943} C_VEL
LIN {X 0,Y 262.436,Z 355.373,A -85,B 0,C 180,E1 -19198.382,E2 -19198.382} C_VEL
LIN {X 0,Y 264.608,Z 351.306,A -85,B 0,C 180,E1 -19199.431,E2 -19199.431} C_VEL
LIN {X 0,Y 266.917,Z 344.579,A -85,B 0,C 180,E1 -19201.334,E2 -19201.334} C_VEL
LIN {X 0,Y 268.617,Z 336.797,A -85,B 0,C 180,E1 -19203.68,E2 -19203.68} C_VEL
LIN {X 0,Y 269.619,Z 329.571,A -85,B 0,C 180,E1 -19206.093,E2 -19206.093} C_VEL
LIN {X 0,Y 270.132,Z 324.334,A -85,B 0,C 180,E1 -19208.076,E2 -19208.076} C_VEL
LIN {X 0,Y 270.359,Z 320.643,A -85,B 0,C 180,E1 -19209.749,E2 -19209.749} C_VEL
LIN {X 0,Y 270.362,Z 318.325,A -85,B 0,C 180,E1 -19211.075,E2 -19211.075} C_VEL
LIN {X 0,Y 269.948,Z 316.04,A -85,B 0,C 180,E1 -19213.2,E2 -19213.2} C_VEL
LIN {X 0,Y 269.779,Z 314.581,A -85,B 0,C 180,E1 -19215.301,E2 -19215.301} C_VEL
LIN {X 0,Y 269.913,Z 313.826,A -85,B 0,C 180,E1 -19217.391,E2 -19217.391} C_VEL
LIN {X 0,Y 270.33,Z 313.801,A -85,B 0,C 180,E1 -19219.462,E2 -19219.462} C_VEL
LIN {X 0,Y 270.917,Z 314.596,A -85,B 0,C 180,E1 -19221.494,E2 -19221.494} C_VEL
LIN {X 0,Y 271.847,Z 317.15,A -85,B 0,C 180,E1 -19224.381,E2 -19224.381} C_VEL
LIN {X 0,Y 272.259,Z 319.704,A -85,B 0,C 180,E1 -19226.16,E2 -19226.16} C_VEL
LIN {X 0,Y 272.617,Z 323.527,A -85,B 0,C 180,E1 -19228.293,E2 -19228.293} C_VEL
LIN {X 0,Y 272.606,Z 328.641,A -85,B 0,C 180,E1 -19230.67,E2 -19230.67} C_VEL
LIN {X 0,Y 272.467,Z 330.121,A -85,B 0,C 180,E1 -19231.283,E2 -19231.283} C_VEL
LIN {X 0,Y 266.954,Z 338.96,A -85,B 0,C 180,E1 -19233.413,E2 -19233.413} C_VEL
LIN {X 0,Y 262.36,Z 345.686,A -85,B 0,C 180,E1 -19235.468,E2 -19235.468} C_VEL
LIN {X 0,Y 256.914,Z 352.942,A -85,B 0,C 180,E1 -19238.328,E2 -19238.328} C_VEL
LIN {X 0,Y 253.34,Z 357.214,A -85,B 0,C 180,E1 -19240.555,E2 -19240.555} C_VEL
LIN {X 0,Y 249.16,Z 361.532,A -85,B 0,C 180,E1 -19243.616,E2 -19243.616} C_VEL
LIN {X 0,Y 245.904,Z 364.33,A -85,B 0,C 180,E1 -19246.783,E2 -19246.783} C_VEL
LIN {X 0,Y 244.367,Z 365.224,A -85,B 0,C 180,E1 -19248.386,E2 -19248.386} C_VEL
LIN {X 0,Y 242.596,Z 365.811,A -85,B 0,C 180,E1 -19251.672,E2 -19251.672} C_VEL
LIN {X 0,Y 241.291,Z 364.996,A -85,B 0,C 180,E1 -19254.987,E2 -19254.987} C_VEL
LIN {X 0,Y 240.323,Z 362.715,A -85,B 0,C 180,E1 -19258.324,E2 -19258.324} C_VEL
LIN {X 0,Y 240.118,Z 358.83,A -85,B 0,C 180,E1 -19261.677,E2 -19261.677} C_VEL
LIN {X 0,Y 240.106,Z 354.803,A -85,B 0,C 180,E1 -19264.197,E2 -19264.197} C_VEL
LIN {X 0,Y 240.309,Z 349.684,A -85,B 0,C 180,E1 -19266.718,E2 -19266.718} C_VEL
LIN {X 0,Y 240.712,Z 343.354,A -85,B 0,C 180,E1 -19269.241,E2 -19269.241} C_VEL
LIN {X 0,Y 241.326,Z 335.592,A -85,B 0,C 180,E1 -19271.763,E2 -19271.763} C_VEL
LIN {X 0,Y 242.306,Z 326.058,A -85,B 0,C 180,E1 -19274.273,E2 -19274.273} C_VEL
LIN {X 0,Y 243.354,Z 315.401,A -85,B 0,C 180,E1 -19276.57,E2 -19276.57} C_VEL
LIN {X 0,Y 244.514,Z 303.405,A -85,B 0,C 180,E1 -19278.649,E2 -19278.649} C_VEL
LIN {X 0,Y 245.714,Z 291.667,A -85,B 0,C 180,E1 -19280.292,E2 -19280.292} C_VEL
LIN {X 0,Y 244.521,Z 283.576,A -85,B 0,C 180,E1 -19281.277,E2 -19281.277} C_VEL
LIN {X 0,Y 242.355,Z 270.94,A -85,B 0,C 180,E1 -19282.576,E2 -19282.576} C_VEL
LIN {X 0,Y 240.483,Z 258.929,A -85,B 0,C 180,E1 -19283.579,E2 -19283.579} C_VEL
LIN {X 0,Y 240.489,Z 258.531,A -85,B 0,C 180,E1 -19284.151,E2 -19284.151} C_VEL
LIN {X 0,Y 241.048,Z 258.458,A -85,B 0,C 180,E1 -19288.992,E2 -19288.992} C_VEL
LIN {X 0,Y 241.561,Z 258.393,A -85,B 0,C 180,E1 -19293.559,E2 -19293.559} C_VEL
LIN {X 0,Y 241.783,Z 258.367,A -85,B 0,C 180,E1 -19295.546,E2 -19295.546} C_VEL
LIN {X 0,Y 241.952,Z 258.345,A -85,B 0,C 180,E1 -19298.346,E2 -19298.346} C_VEL
LIN {X 0,Y 241.932,Z 258.346,A -85,B 0,C 180,E1 -19301.924,E2 -19301.924} C_VEL
LIN {X 0,Y 241.924,Z 258.35,A -85,B 0,C 180,E1 -19306.575,E2 -19306.575} C_VEL
LIN {X 0,Y 241.995,Z 258.34,A -85,B 0,C 180,E1 -19311.641,E2 -19311.641} C_VEL
LIN {X 0,Y 241.982,Z 258.342,A -85,B 0,C 180,E1 -19314.488,E2 -19314.488} C_VEL
LIN {X 0,Y 241.957,Z 258.346,A -85,B 0,C 180,E1 -19318.477,E2 -19318.477} C_VEL
LIN {X 0,Y 241.977,Z 258.344,A -85,B 0,C 180,E1 -19322.308,E2 -19322.308} C_VEL
LIN {X 0,Y 242.04,Z 258.335,A -85,B 0,C 180,E1 -19326.014,E2 -19326.014} C_VEL
LIN {X 0,Y 242.039,Z 258.334,A -85,B 0,C 180,E1 -19329.608,E2 -19329.608} C_VEL
LIN {X 0,Y 242.167,Z 258.315,A -85,B 0,C 180,E1 -19333.278,E2 -19333.278} C_VEL
LIN {X 0,Y 242.183,Z 258.318,A -85,B 0,C 180,E1 -19338.279,E2 -19338.279} C_VEL
LIN {X 0,Y 242.387,Z 258.294,A -85,B 0,C 180,E1 -19341.664,E2 -19341.664} C_VEL
LIN {X 0,Y 242.402,Z 258.291,A -85,B 0,C 180,E1 -19343.34,E2 -19343.34} C_VEL
LIN {X 0,Y 242.619,Z 258.264,A -85,B 0,C 180,E1 -19348.34,E2 -19348.34} C_VEL
LIN {X 0,Y 242.626,Z 258.436,A -85,B 0,C 180,E1 -19351.245,E2 -19351.245} C_VEL
LIN {X 0,Y 242.857,Z 264.189,A -85,B 0,C 180,E1 -19354.98,E2 -19354.98} C_VEL
LIN {X 0,Y 242.384,Z 271.553,A -85,B 0,C 180,E1 -19359.651,E2 -19359.651} C_VEL
LIN {X 0,Y 242.003,Z 277.545,A -85,B 0,C 180,E1 -19363.434,E2 -19363.434} C_VEL
LIN {X 0,Y 241.812,Z 281.32,A -85,B 0,C 180,E1 -19365.796,E2 -19365.796} C_VEL
LIN {X 0,Y 243.753,Z 291.459,A -85,B 0,C 180,E1 -19366.55,E2 -19366.55} C_VEL
LIN {X 0,Y 245.31,Z 301.277,A -85,B 0,C 180,E1 -19367.507,E2 -19367.507} C_VEL
LIN {X 0,Y 246.544,Z 311.031,A -85,B 0,C 180,E1 -19368.704,E2 -19368.704} C_VEL
LIN {X 0,Y 245.531,Z 320.616,A -85,B 0,C 180,E1 -19370.089,E2 -19370.089} C_VEL
LIN {X 0,Y 244.532,Z 328.397,A -85,B 0,C 180,E1 -19371.496,E2 -19371.496} C_VEL
LIN {X 0,Y 243.691,Z 334.697,A -85,B 0,C 180,E1 -19372.868,E2 -19372.868} C_VEL
LIN {X 0,Y 242.927,Z 340.399,A -85,B 0,C 180,E1 -19374.347,E2 -19374.347} C_VEL
LIN {X 0,Y 242.014,Z 346.525,A -85,B 0,C 180,E1 -19376.285,E2 -19376.285} C_VEL
LIN {X 0,Y 241.433,Z 350.4,A -85,B 0,C 180,E1 -19377.759,E2 -19377.759} C_VEL
LIN {X 0,Y 240.878,Z 354.621,A -85,B 0,C 180,E1 -19379.736,E2 -19379.736} C_VEL
LIN {X 0,Y 240.326,Z 358.324,A -85,B 0,C 180,E1 -19381.998,E2 -19381.998} C_VEL
LIN {X 0,Y 240.02,Z 360.519,A -85,B 0,C 180,E1 -19383.803,E2 -19383.803} C_VEL
LIN {X 0,Y 239.869,Z 362.255,A -85,B 0,C 180,E1 -19385.873,E2 -19385.873} C_VEL
LIN {X 0,Y 239.916,Z 363.214,A -85,B 0,C 180,E1 -19387.964,E2 -19387.964} C_VEL
LIN {X 0,Y 240.237,Z 363.332,A -85,B 0,C 180,E1 -19390.481,E2 -19390.481} C_VEL
LIN {X 0,Y 240.906,Z 362.262,A -85,B 0,C 180,E1 -19393.169,E2 -19393.169} C_VEL
LIN {X 0,Y 241.823,Z 359.9,A -85,B 0,C 180,E1 -19395.772,E2 -19395.772} C_VEL
LIN {X 0,Y 242.561,Z 357.743,A -85,B 0,C 180,E1 -19397.411,E2 -19397.411} C_VEL
LIN {X 0,Y 243.938,Z 353.543,A -85,B 0,C 180,E1 -19399.744,E2 -19399.744} C_VEL
LIN {X 0,Y 245.455,Z 348.285,A -85,B 0,C 180,E1 -19401.943,E2 -19401.943} C_VEL
LIN {X 0,Y 246.853,Z 343.347,A -85,B 0,C 180,E1 -19403.596,E2 -19403.596} C_VEL
LIN {X 0,Y 248.372,Z 337.725,A -85,B 0,C 180,E1 -19405.144,E2 -19405.144} C_VEL
LIN {X 0,Y 250.162,Z 330.318,A -85,B 0,C 180,E1 -19406.807,E2 -19406.807} C_VEL
LIN {X 0,Y 252.12,Z 320.937,A -85,B 0,C 180,E1 -19408.488,E2 -19408.488} C_VEL
LIN {X 0,Y 252.15,Z 316.667,A -85,B 0,C 180,E1 -19409.192,E2 -19409.192} C_VEL
LIN {X 0,Y 251.255,Z 309.039,A -85,B 0,C 180,E1 -19410.438,E2 -19410.438} C_VEL
LIN {X 0,Y 249.367,Z 299.53,A -85,B 0,C 180,E1 -19411.831,E2 -19411.831} C_VEL
LIN {X 0,Y 245.797,Z 287.796,A -85,B 0,C 180,E1 -19413.377,E2 -19413.377} C_VEL
LIN {X 0,Y 244.177,Z 283.141,A -85,B 0,C 180,E1 -19413.942,E2 -19413.942} C_VEL
LIN {X 0,Y 244.835,Z 277.021,A -85,B 0,C 180,E1 -19418.089,E2 -19418.089} C_VEL
LIN {X 0,Y 245.057,Z 274.457,A -85,B 0,C 180,E1 -19419.87,E2 -19419.87} C_VEL
LIN {X 0,Y 244.788,Z 270.95,A -85,B 0,C 180,E1 -19422.454,E2 -19422.454} C_VEL
LIN {X 0,Y 244.1,Z 266.565,A -85,B 0,C 180,E1 -19425.834,E2 -19425.834} C_VEL
LIN {X 0,Y 243.033,Z 261.524,A -85,B 0,C 180,E1 -19430.008,E2 -19430.008} C_VEL
LIN {X 0,Y 242.387,Z 258.293,A -85,B 0,C 180,E1 -19432.921,E2 -19432.921} C_VEL
LIN {X 0,Y 242.637,Z 258.263,A -85,B 0,C 180,E1 -19438.34,E2 -19438.34} C_VEL
LIN {X 0,Y 242.637,Z 258.26,A -85,B 0,C 180,E1 -19441.66,E2 -19441.66} C_VEL
LIN {X 0,Y 242.41,Z 258.288,A -85,B 0,C 180,E1 -19446.659,E2 -19446.659} C_VEL
LIN {X 0,Y 242.269,Z 258.308,A -85,B 0,C 180,E1 -19450.023,E2 -19450.023} C_VEL
LIN {X 0,Y 242.168,Z 258.319,A -85,B 0,C 180,E1 -19455.141,E2 -19455.141} C_VEL
LIN {X 0,Y 242.074,Z 258.327,A -85,B 0,C 180,E1 -19458.624,E2 -19458.624} C_VEL
LIN {X 0,Y 242.008,Z 258.338,A -85,B 0,C 180,E1 -19462.18,E2 -19462.18} C_VEL
LIN {X 0,Y 242.068,Z 258.332,A -85,B 0,C 180,E1 -19465.838,E2 -19465.838} C_VEL
LIN {X 0,Y 242.031,Z 258.332,A -85,B 0,C 180,E1 -19469.58,E2 -19469.58} C_VEL
LIN {X 0,Y 241.989,Z 258.342,A -85,B 0,C 180,E1 -19473.491,E2 -19473.491} C_VEL
LIN {X 0,Y 241.978,Z 258.336,A -85,B 0,C 180,E1 -19476.526,E2 -19476.526} C_VEL
LIN {X 0,Y 241.291,Z 258.428,A -85,B 0,C 180,E1 -19477.915,E2 -19477.915} C_VEL
LIN {X 0,Y 238.436,Z 258.781,A -85,B 0,C 180,E1 -19480.183,E2 -19480.183} C_VEL
LIN {X 0,Y 236.071,Z 259.079,A -85,B 0,C 180,E1 -19482.03,E2 -19482.03} C_VEL
LIN {X 0,Y 235.125,Z 259.197,A -85,B 0,C 180,E1 -19483.464,E2 -19483.464} C_VEL
LIN {X 0,Y 235.085,Z 259.201,A -85,B 0,C 180,E1 -19483.948,E2 -19483.948} C_VEL
LIN {X 0,Y 235.137,Z 259.341,A -85,B 0,C 180,E1 -19484.455,E2 -19484.455} C_VEL
LIN {X 0,Y 236.064,Z 264.334,A -85,B 0,C 180,E1 -19489.082,E2 -19489.082} C_VEL
LIN {X 0,Y 236.613,Z 267.536,A -85,B 0,C 180,E1 -19491.91,E2 -19491.91} C_VEL
LIN {X 0,Y 237.335,Z 274.217,A -85,B 0,C 180,E1 -19494.73,E2 -19494.73} C_VEL
LIN {X 0,Y 237.722,Z 285.139,A -85,B 0,C 180,E1 -19498.413,E2 -19498.413} C_VEL
LIN {X 0,Y 238.283,Z 296.698,A -85,B 0,C 180,E1 -19501.842,E2 -19501.842} C_VEL
LIN {X 0,Y 238.34,Z 297.833,A -85,B 0,C 180,E1 -19502.112,E2 -19502.112} C_VEL
LIN {X 0,Y 242.05,Z 311.681,A -85,B 0,C 180,E1 -19503.48,E2 -19503.48} C_VEL
LIN {X 0,Y 242.499,Z 316.866,A -85,B 0,C 180,E1 -19503.976,E2 -19503.976} C_VEL
LIN {X 0,Y 242.672,Z 329.493,A -85,B 0,C 180,E1 -19505.35,E2 -19505.35} C_VEL
LIN {X 0,Y 242.586,Z 337.89,A -85,B 0,C 180,E1 -19506.525,E2 -19506.525} C_VEL
LIN {X 0,Y 242.307,Z 342.121,A -85,B 0,C 180,E1 -19507.174,E2 -19507.174} C_VEL
LIN {X 0,Y 240.467,Z 351.591,A -85,B 0,C 180,E1 -19508.797,E2 -19508.797} C_VEL
LIN {X 0,Y 238.811,Z 358.811,A -85,B 0,C 180,E1 -19510.345,E2 -19510.345} C_VEL
LIN {X 0,Y 237.604,Z 364.753,A -85,B 0,C 180,E1 -19511.906,E2 -19511.906} C_VEL
LIN {X 0,Y 236.088,Z 371.306,A -85,B 0,C 180,E1 -19514.017,E2 -19514.017} C_VEL
LIN {X 0,Y 234.741,Z 376.603,A -85,B 0,C 180,E1 -19516.142,E2 -19516.142} C_VEL
LIN {X 0,Y 233.77,Z 381.571,A -85,B 0,C 180,E1 -19518.731,E2 -19518.731} C_VEL
LIN {X 0,Y 233.184,Z 385.084,A -85,B 0,C 180,E1 -19521.333,E2 -19521.333} C_VEL
LIN {X 0,Y 232.997,Z 386.778,A -85,B 0,C 180,E1 -19523.07,E2 -19523.07} C_VEL
LIN {X 0,Y 232.881,Z 387.876,A -85,B 0,C 180,E1 -19524.806,E2 -19524.806} C_VEL
LIN {X 0,Y 232.957,Z 388.488,A -85,B 0,C 180,E1 -19526.541,E2 -19526.541} C_VEL
LIN {X 0,Y 233.054,Z 388.624,A -85,B 0,C 180,E1 -19528.272,E2 -19528.272} C_VEL
LIN {X 0,Y 233.167,Z 388.276,A -85,B 0,C 180,E1 -19530,E2 -19530} C_VEL
LIN {X 0,Y 233.142,Z 386.637,A -85,B 0,C 180,E1 -19532.592,E2 -19532.592} C_VEL
LIN {X 0,Y 233.111,Z 386.519,A -85,B 0,C 180,E1 -19533.025,E2 -19533.025} C_VEL
LIN {X 0,Y 232.937,Z 387.657,A -85,B 0,C 180,E1 -19535.344,E2 -19535.344} C_VEL
LIN {X 0,Y 233.159,Z 388.11,A -85,B 0,C 180,E1 -19538.669,E2 -19538.669} C_VEL
LIN {X 0,Y 234.172,Z 387.205,A -85,B 0,C 180,E1 -19542.128,E2 -19542.128} C_VEL
LIN {X 0,Y 236.113,Z 384.935,A -85,B 0,C 180,E1 -19545.539,E2 -19545.539} C_VEL
LIN {X 0,Y 239.24,Z 381.228,A -85,B 0,C 180,E1 -19548.853,E2 -19548.853} C_VEL
LIN {X 0,Y 241.922,Z 377.557,A -85,B 0,C 180,E1 -19551.293,E2 -19551.293} C_VEL
LIN {X 0,Y 245.256,Z 373.01,A -85,B 0,C 180,E1 -19553.652,E2 -19553.652} C_VEL
LIN {X 0,Y 250.812,Z 365.472,A -85,B 0,C 180,E1 -19556.637,E2 -19556.637} C_VEL
LIN {X 0,Y 256.406,Z 357.384,A -85,B 0,C 180,E1 -19559.113,E2 -19559.113} C_VEL
LIN {X 0,Y 259.355,Z 352.291,A -85,B 0,C 180,E1 -19560.537,E2 -19560.537} C_VEL
LIN {X 0,Y 261.699,Z 345.933,A -85,B 0,C 180,E1 -19562.487,E2 -19562.487} C_VEL
LIN {X 0,Y 263.658,Z 338.46,A -85,B 0,C 180,E1 -19564.967,E2 -19564.967} C_VEL
LIN {X 0,Y 264.989,Z 331.406,A -85,B 0,C 180,E1 -19567.59,E2 -19567.59} C_VEL
LIN {X 0,Y 265.755,Z 326.186,A -85,B 0,C 180,E1 -19569.922,E2 -19569.922} C_VEL
LIN {X 0,Y 265.945,Z 323.776,A -85,B 0,C 180,E1 -19571.351,E2 -19571.351} C_VEL
LIN {X 0,Y 265.706,Z 321.606,A -85,B 0,C 180,E1 -19573.449,E2 -19573.449} C_VEL
LIN {X 0,Y 265.658,Z 319.846,A -85,B 0,C 180,E1 -19576.541,E2 -19576.541} C_VEL
LIN {X 0,Y 265.939,Z 319.501,A -85,B 0,C 180,E1 -19578.648,E2 -19578.648} C_VEL
LIN {X 0,Y 266.397,Z 319.902,A -85,B 0,C 180,E1 -19580.716,E2 -19580.716} C_VEL
LIN {X 0,Y 266.819,Z 321.159,A -85,B 0,C 180,E1 -19582.712,E2 -19582.712} C_VEL
LIN {X 0,Y 267.262,Z 323.066,A -85,B 0,C 180,E1 -19584.654,E2 -19584.654} C_VEL
LIN {X 0,Y 267.499,Z 326.838,A -85,B 0,C 180,E1 -19587.219,E2 -19587.219} C_VEL
LIN {X 0,Y 267.363,Z 330.808,A -85,B 0,C 180,E1 -19589.355,E2 -19589.355} C_VEL
LIN {X 0,Y 267.138,Z 332.714,A -85,B 0,C 180,E1 -19590.249,E2 -19590.249} C_VEL
LIN {X 0,Y 265.413,Z 335.765,A -85,B 0,C 180,E1 -19591.102,E2 -19591.102} C_VEL
LIN {X 0,Y 260.199,Z 343.086,A -85,B 0,C 180,E1 -19593.101,E2 -19593.101} C_VEL
LIN {X 0,Y 254.779,Z 350.074,A -85,B 0,C 180,E1 -19595.558,E2 -19595.558} C_VEL
LIN {X 0,Y 250.586,Z 354.968,A -85,B 0,C 180,E1 -19597.752,E2 -19597.752} C_VEL
LIN {X 0,Y 245.698,Z 360.069,A -85,B 0,C 180,E1 -19600.795,E2 -19600.795} C_VEL
LIN {X 0,Y 242.492,Z 362.879,A -85,B 0,C 180,E1 -19603.153,E2 -19603.153} C_VEL
LIN {X 0,Y 239.064,Z 365.319,A -85,B 0,C 180,E1 -19606.398,E2 -19606.398} C_VEL
LIN {X 0,Y 237.472,Z 366.025,A -85,B 0,C 180,E1 -19608.044,E2 -19608.044} C_VEL
LIN {X 0,Y 235.596,Z 366.324,A -85,B 0,C 180,E1 -19611.422,E2 -19611.422} C_VEL
LIN {X 0,Y 234.233,Z 365.22,A -85,B 0,C 180,E1 -19614.836,E2 -19614.836} C_VEL
LIN {X 0,Y 233.247,Z 362.616,A -85,B 0,C 180,E1 -19618.274,E2 -19618.274} C_VEL
LIN {X 0,Y 233.047,Z 358.483,A -85,B 0,C 180,E1 -19621.728,E2 -19621.728} C_VEL
LIN {X 0,Y 233.015,Z 354.222,A -85,B 0,C 180,E1 -19624.325,E2 -19624.325} C_VEL
LIN {X 0,Y 233.305,Z 347.824,A -85,B 0,C 180,E1 -19627.356,E2 -19627.356} C_VEL
LIN {X 0,Y 233.803,Z 340.985,A -85,B 0,C 180,E1 -19629.953,E2 -19629.953} C_VEL
LIN {X 0,Y 234.461,Z 332.621,A -85,B 0,C 180,E1 -19632.552,E2 -19632.552} C_VEL
LIN {X 0,Y 235.546,Z 322.362,A -85,B 0,C 180,E1 -19635.134,E2 -19635.134} C_VEL
LIN {X 0,Y 236.546,Z 311.921,A -85,B 0,C 180,E1 -19637.284,E2 -19637.284} C_VEL
LIN {X 0,Y 237.953,Z 299.094,A -85,B 0,C 180,E1 -19639.407,E2 -19639.407} C_VEL
LIN {X 0,Y 238.629,Z 291.38,A -85,B 0,C 180,E1 -19640.472,E2 -19640.472} C_VEL
LIN {X 0,Y 236.335,Z 277.805,A -85,B 0,C 180,E1 -19642.095,E2 -19642.095} C_VEL
LIN {X 0,Y 233.939,Z 263.533,A -85,B 0,C 180,E1 -19643.417,E2 -19643.417} C_VEL
LIN {X 0,Y 233.399,Z 259.414,A -85,B 0,C 180,E1 -19643.75,E2 -19643.75} C_VEL
LIN {X 0,Y 233.975,Z 259.339,A -85,B 0,C 180,E1 -19648.725,E2 -19648.725} C_VEL
LIN {X 0,Y 234.43,Z 259.282,A -85,B 0,C 180,E1 -19652.92,E2 -19652.92} C_VEL
LIN {X 0,Y 234.795,Z 259.237,A -85,B 0,C 180,E1 -19656.774,E2 -19656.774} C_VEL
LIN {X 0,Y 234.889,Z 259.227,A -85,B 0,C 180,E1 -19658.927,E2 -19658.927} C_VEL
LIN {X 0,Y 234.881,Z 259.228,A -85,B 0,C 180,E1 -19663.488,E2 -19663.488} C_VEL
LIN {X 0,Y 234.877,Z 259.227,A -85,B 0,C 180,E1 -19666.511,E2 -19666.511} C_VEL
LIN {X 0,Y 234.92,Z 259.224,A -85,B 0,C 180,E1 -19671.078,E2 -19671.078} C_VEL
LIN {X 0,Y 234.928,Z 259.221,A -85,B 0,C 180,E1 -19675.361,E2 -19675.361} C_VEL
LIN {X 0,Y 234.903,Z 259.222,A -85,B 0,C 180,E1 -19679.428,E2 -19679.428} C_VEL
LIN {X 0,Y 234.972,Z 259.215,A -85,B 0,C 180,E1 -19683.806,E2 -19683.806} C_VEL
LIN {X 0,Y 235.001,Z 259.211,A -85,B 0,C 180,E1 -19688.968,E2 -19688.968} C_VEL
LIN {X 0,Y 235.1,Z 259.195,A -85,B 0,C 180,E1 -19693.059,E2 -19693.059} C_VEL
LIN {X 0,Y 235.117,Z 259.196,A -85,B 0,C 180,E1 -19697.922,E2 -19697.922} C_VEL
LIN {X 0,Y 235.321,Z 259.174,A -85,B 0,C 180,E1 -19701.412,E2 -19701.412} C_VEL
LIN {X 0,Y 235.355,Z 259.169,A -85,B 0,C 180,E1 -19703.14,E2 -19703.14} C_VEL
LIN {X 0,Y 235.578,Z 259.141,A -85,B 0,C 180,E1 -19708.29,E2 -19708.29} C_VEL
LIN {X 0,Y 235.575,Z 259.326,A -85,B 0,C 180,E1 -19710.854,E2 -19710.854} C_VEL
LIN {X 0,Y 235.874,Z 264.412,A -85,B 0,C 180,E1 -19714.272,E2 -19714.272} C_VEL
LIN {X 0,Y 235.484,Z 271.128,A -85,B 0,C 180,E1 -19718.582,E2 -19718.582} C_VEL
LIN {X 0,Y 235.018,Z 277.937,A -85,B 0,C 180,E1 -19722.96,E2 -19722.96} C_VEL
LIN {X 0,Y 234.827,Z 281.59,A -85,B 0,C 180,E1 -19725.292,E2 -19725.292} C_VEL
LIN {X 0,Y 237.008,Z 293.144,A -85,B 0,C 180,E1 -19726.222,E2 -19726.222} C_VEL
LIN {X 0,Y 238.649,Z 303.882,A -85,B 0,C 180,E1 -19727.341,E2 -19727.341} C_VEL
LIN {X 0,Y 239.569,Z 312.576,A -85,B 0,C 180,E1 -19728.49,E2 -19728.49} C_VEL
LIN {X 0,Y 238.459,Z 321.962,A -85,B 0,C 180,E1 -19729.929,E2 -19729.929} C_VEL
LIN {X 0,Y 237.533,Z 328.985,A -85,B 0,C 180,E1 -19731.25,E2 -19731.25} C_VEL
LIN {X 0,Y 236.542,Z 336.26,A -85,B 0,C 180,E1 -19732.918,E2 -19732.918} C_VEL
LIN {X 0,Y 235.586,Z 342.589,A -85,B 0,C 180,E1 -19734.686,E2 -19734.686} C_VEL
LIN {X 0,Y 234.75,Z 348.406,A -85,B 0,C 180,E1 -19736.684,E2 -19736.684} C_VEL
LIN {X 0,Y 233.864,Z 354.44,A -85,B 0,C 180,E1 -19739.366,E2 -19739.366} C_VEL
LIN {X 0,Y 233.32,Z 358.146,A -85,B 0,C 180,E1 -19741.598,E2 -19741.598} C_VEL
LIN {X 0,Y 232.915,Z 360.964,A -85,B 0,C 180,E1 -19743.933,E2 -19743.933} C_VEL
LIN {X 0,Y 232.797,Z 362.29,A -85,B 0,C 180,E1 -19745.401,E2 -19745.401} C_VEL
LIN {X 0,Y 232.778,Z 363.315,A -85,B 0,C 180,E1 -19747.145,E2 -19747.145} C_VEL
LIN {X 0,Y 232.958,Z 363.865,A -85,B 0,C 180,E1 -19749.312,E2 -19749.312} C_VEL
LIN {X 0,Y 233.367,Z 363.623,A -85,B 0,C 180,E1 -19751.494,E2 -19751.494} C_VEL
LIN {X 0,Y 234.024,Z 362.439,A -85,B 0,C 180,E1 -19753.883,E2 -19753.883} C_VEL
LIN {X 0,Y 235.077,Z 359.853,A -85,B 0,C 180,E1 -19756.557,E2 -19756.557} C_VEL
LIN {X 0,Y 235.844,Z 357.745,A -85,B 0,C 180,E1 -19758.158,E2 -19758.158} C_VEL
LIN {X 0,Y 237.247,Z 353.783,A -85,B 0,C 180,E1 -19760.372,E2 -19760.372} C_VEL
LIN {X 0,Y 238.852,Z 348.571,A -85,B 0,C 180,E1 -19762.603,E2 -19762.603} C_VEL
LIN {X 0,Y 240.244,Z 343.956,A -85,B 0,C 180,E1 -19764.192,E2 -19764.192} C_VEL
LIN {X 0,Y 241.945,Z 337.967,A -85,B 0,C 180,E1 -19765.88,E2 -19765.88} C_VEL
LIN {X 0,Y 243.751,Z 330.921,A -85,B 0,C 180,E1 -19767.496,E2 -19767.496} C_VEL
LIN {X 0,Y 245.668,Z 322.166,A -85,B 0,C 180,E1 -19769.119,E2 -19769.119} C_VEL
LIN {X 0,Y 245.765,Z 318.885,A -85,B 0,C 180,E1 -19769.693,E2 -19769.693} C_VEL
LIN {X 0,Y 244.971,Z 311.131,A -85,B 0,C 180,E1 -19771.044,E2 -19771.044} C_VEL
LIN {X 0,Y 243.592,Z 303.402,A -85,B 0,C 180,E1 -19772.274,E2 -19772.274} C_VEL
LIN {X 0,Y 241.297,Z 294.706,A -85,B 0,C 180,E1 -19773.547,E2 -19773.547} C_VEL
LIN {X 0,Y 238.519,Z 286.54,A -85,B 0,C 180,E1 -19774.648,E2 -19774.648} C_VEL
LIN {X 0,Y 237.476,Z 283.499,A -85,B 0,C 180,E1 -19775.056,E2 -19775.056} C_VEL
LIN {X 0,Y 238.197,Z 277.491,A -85,B 0,C 180,E1 -19779.264,E2 -19779.264} C_VEL
LIN {X 0,Y 238.142,Z 273.863,A -85,B 0,C 180,E1 -19781.948,E2 -19781.948} C_VEL
LIN {X 0,Y 237.511,Z 269.506,A -85,B 0,C 180,E1 -19785.432,E2 -19785.432} C_VEL
LIN {X 0,Y 236.487,Z 264.474,A -85,B 0,C 180,E1 -19789.728,E2 -19789.728} C_VEL
LIN {X 0,Y 235.718,Z 260.692,A -85,B 0,C 180,E1 -19793.15,E2 -19793.15} C_VEL
LIN {X 0,Y 235.223,Z 259.185,A -85,B 0,C 180,E1 -19794.642,E2 -19794.642} C_VEL
LIN {X 0,Y 235.596,Z 259.139,A -85,B 0,C 180,E1 -19798.29,E2 -19798.29} C_VEL
LIN {X 0,Y 235.596,Z 259.137,A -85,B 0,C 180,E1 -19801.709,E2 -19801.709} C_VEL
LIN {X 0,Y 235.361,Z 259.167,A -85,B 0,C 180,E1 -19806.86,E2 -19806.86} C_VEL
LIN {X 0,Y 235.216,Z 259.184,A -85,B 0,C 180,E1 -19810.327,E2 -19810.327} C_VEL
LIN {X 0,Y 235.115,Z 259.195,A -85,B 0,C 180,E1 -19815.606,E2 -19815.606} C_VEL
LIN {X 0,Y 235.009,Z 259.208,A -85,B 0,C 180,E1 -19819.205,E2 -19819.205} C_VEL
LIN {X 0,Y 234.954,Z 259.22,A -85,B 0,C 180,E1 -19822.883,E2 -19822.883} C_VEL
LIN {X 0,Y 234.97,Z 259.212,A -85,B 0,C 180,E1 -19826.657,E2 -19826.657} C_VEL
LIN {X 0,Y 234.933,Z 259.221,A -85,B 0,C 180,E1 -19830.567,E2 -19830.567} C_VEL
LIN {X 0,Y 234.96,Z 259.212,A -85,B 0,C 180,E1 -19834.633,E2 -19834.633} C_VEL
LIN {X 0,Y 234.942,Z 259.218,A -85,B 0,C 180,E1 -19838.944,E2 -19838.944} C_VEL
LIN {X 0,Y 235.085,Z 259.201,A -85,B 0,C 180,E1 -19843.948,E2 -19843.948} C_VEL
LIN {X 0,Y 234.886,Z 259.849,A -85,B 0,C 180,E1 -19844.898,E2 -19844.898} C_VEL
LIN {X 0,Y 233.337,Z 261.988,A -85,B 0,C 180,E1 -19846.721,E2 -19846.721} C_VEL
LIN {X 0,Y 231.828,Z 263.866,A -85,B 0,C 180,E1 -19848.035,E2 -19848.035} C_VEL
LIN {X 0,Y 230.57,Z 266.525,A -85,B 0,C 180,E1 -19849.351,E2 -19849.351} C_VEL
LIN {X 0,Y 230.14,Z 269.25,A -85,B 0,C 180,E1 -19850.685,E2 -19850.685} C_VEL
LIN {X 0,Y 230.282,Z 270.126,A -85,B 0,C 180,E1 -19851.134,E2 -19851.134} C_VEL
LIN {X 0,Y 230.939,Z 274.29,A -85,B 0,C 180,E1 -19853.038,E2 -19853.038} C_VEL
LIN {X 0,Y 231.205,Z 279.675,A -85,B 0,C 180,E1 -19855.158,E2 -19855.158} C_VEL
LIN {X 0,Y 231.489,Z 289.682,A -85,B 0,C 180,E1 -19858.588,E2 -19858.588} C_VEL
LIN {X 0,Y 231.826,Z 297.636,A -85,B 0,C 180,E1 -19860.957,E2 -19860.957} C_VEL
LIN {X 0,Y 235.514,Z 311.071,A -85,B 0,C 180,E1 -19862.39,E2 -19862.39} C_VEL
LIN {X 0,Y 236.451,Z 316.952,A -85,B 0,C 180,E1 -19863.047,E2 -19863.047} C_VEL
LIN {X 0,Y 236.38,Z 329.206,A -85,B 0,C 180,E1 -19864.419,E2 -19864.419} C_VEL
LIN {X 0,Y 236.15,Z 338.867,A -85,B 0,C 180,E1 -19865.845,E2 -19865.845} C_VEL
LIN {X 0,Y 235.827,Z 343.003,A -85,B 0,C 180,E1 -19866.51,E2 -19866.51} C_VEL
LIN {X 0,Y 234.174,Z 351.116,A -85,B 0,C 180,E1 -19867.967,E2 -19867.967} C_VEL
LIN {X 0,Y 232.298,Z 358.691,A -85,B 0,C 180,E1 -19869.633,E2 -19869.633} C_VEL
LIN {X 0,Y 230.861,Z 365.003,A -85,B 0,C 180,E1 -19871.359,E2 -19871.359} C_VEL
LIN {X 0,Y 229.247,Z 371.444,A -85,B 0,C 180,E1 -19873.526,E2 -19873.526} C_VEL
LIN {X 0,Y 227.836,Z 376.629,A -85,B 0,C 180,E1 -19875.714,E2 -19875.714} C_VEL
LIN {X 0,Y 226.782,Z 381.469,A -85,B 0,C 180,E1 -19878.379,E2 -19878.379} C_VEL
LIN {X 0,Y 226.136,Z 384.859,A -85,B 0,C 180,E1 -19881.061,E2 -19881.061} C_VEL
LIN {X 0,Y 225.923,Z 386.518,A -85,B 0,C 180,E1 -19882.852,E2 -19882.852} C_VEL
LIN {X 0,Y 225.788,Z 387.728,A -85,B 0,C 180,E1 -19884.905,E2 -19884.905} C_VEL
LIN {X 0,Y 225.868,Z 388.132,A -85,B 0,C 180,E1 -19886.432,E2 -19886.432} C_VEL
LIN {X 0,Y 225.976,Z 388.201,A -85,B 0,C 180,E1 -19888.218,E2 -19888.218} C_VEL
LIN {X 0,Y 226.086,Z 387.788,A -85,B 0,C 180,E1 -19890,E2 -19890} C_VEL
LIN {X 0,Y 226.1,Z 386.854,A -85,B 0,C 180,E1 -19891.782,E2 -19891.782} C_VEL
LIN {X 0,Y 226.018,Z 385.705,A -85,B 0,C 180,E1 -19893.343,E2 -19893.343} C_VEL
LIN {X 0,Y 225.899,Z 386.799,A -85,B 0,C 180,E1 -19895.401,E2 -19895.401} C_VEL
LIN {X 0,Y 226.145,Z 387.573,A -85,B 0,C 180,E1 -19898.94,E2 -19898.94} C_VEL
LIN {X 0,Y 227.21,Z 386.938,A -85,B 0,C 180,E1 -19902.505,E2 -19902.505} C_VEL
LIN {X 0,Y 229.271,Z 384.938,A -85,B 0,C 180,E1 -19906.015,E2 -19906.015} C_VEL
LIN {X 0,Y 232.52,Z 381.594,A -85,B 0,C 180,E1 -19909.42,E2 -19909.42} C_VEL
LIN {X 0,Y 235.351,Z 378.18,A -85,B 0,C 180,E1 -19911.918,E2 -19911.918} C_VEL
LIN {X 0,Y 240.221,Z 372.355,A -85,B 0,C 180,E1 -19915.102,E2 -19915.102} C_VEL
LIN {X 0,Y 245.415,Z 365.938,A -85,B 0,C 180,E1 -19917.734,E2 -19917.734} C_VEL
LIN {X 0,Y 252.111,Z 356.938,A -85,B 0,C 180,E1 -19920.581,E2 -19920.581} C_VEL
LIN {X 0,Y 254.174,Z 353.323,A -85,B 0,C 180,E1 -19921.693,E2 -19921.693} C_VEL
LIN {X 0,Y 256.566,Z 347.525,A -85,B 0,C 180,E1 -19923.658,E2 -19923.658} C_VEL
LIN {X 0,Y 258.431,Z 341.632,A -85,B 0,C 180,E1 -19925.781,E2 -19925.781} C_VEL
LIN {X 0,Y 260.119,Z 335.094,A -85,B 0,C 180,E1 -19928.421,E2 -19928.421} C_VEL
LIN {X 0,Y 260.95,Z 331.24,A -85,B 0,C 180,E1 -19930.27,E2 -19930.27} C_VEL
LIN {X 0,Y 261.177,Z 329.826,A -85,B 0,C 180,E1 -19931.11,E2 -19931.11} C_VEL
LIN {X 0,Y 261.297,Z 328.317,A -85,B 0,C 180,E1 -19932.254,E2 -19932.254} C_VEL
LIN {X 0,Y 261.2,Z 326.524,A -85,B 0,C 180,E1 -19934.393,E2 -19934.393} C_VEL
LIN {X 0,Y 261.264,Z 325.434,A -85,B 0,C 180,E1 -19936.578,E2 -19936.578} C_VEL
LIN {X 0,Y 261.553,Z 325.051,A -85,B 0,C 180,E1 -19938.797,E2 -19938.797} C_VEL
LIN {X 0,Y 261.908,Z 325.595,A -85,B 0,C 180,E1 -19941.095,E2 -19941.095} C_VEL
LIN {X 0,Y 262.309,Z 327.63,A -85,B 0,C 180,E1 -19943.883,E2 -19943.883} C_VEL
LIN {X 0,Y 262.396,Z 330.345,A -85,B 0,C 180,E1 -19946.131,E2 -19946.131} C_VEL
LIN {X 0,Y 262.051,Z 334.114,A -85,B 0,C 180,E1 -19948.469,E2 -19948.469} C_VEL
LIN {X 0,Y 261.487,Z 336.57,A -85,B 0,C 180,E1 -19949.694,E2 -19949.694} C_VEL
LIN {X 0,Y 255.127,Z 344.898,A -85,B 0,C 180,E1 -19952.076,E2 -19952.076} C_VEL
LIN {X 0,Y 250.177,Z 350.743,A -85,B 0,C 180,E1 -19954.188,E2 -19954.188} C_VEL
LIN {X 0,Y 244.274,Z 356.994,A -85,B 0,C 180,E1 -19957.145,E2 -19957.145} C_VEL
LIN {X 0,Y 240.365,Z 360.637,A -85,B 0,C 180,E1 -19959.46,E2 -19959.46} C_VEL
LIN {X 0,Y 235.816,Z 364.155,A -85,B 0,C 180,E1 -19962.661,E2 -19962.661} C_VEL
LIN {X 0,Y 232.229,Z 366.254,A -85,B 0,C 180,E1 -19965.989,E2 -19965.989} C_VEL
LIN {X 0,Y 230.586,Z 366.814,A -85,B 0,C 180,E1 -19967.681,E2 -19967.681} C_VEL
LIN {X 0,Y 228.603,Z 366.77,A -85,B 0,C 180,E1 -19971.158,E2 -19971.158} C_VEL
LIN {X 0,Y 227.178,Z 365.342,A -85,B 0,C 180,E1 -19974.675,E2 -19974.675} C_VEL
LIN {X 0,Y 226.173,Z 362.48,A -85,B 0,C 180,E1 -19978.22,E2 -19978.22} C_VEL
LIN {X 0,Y 225.979,Z 358.004,A -85,B 0,C 180,E1 -19981.782,E2 -19981.782} C_VEL
LIN {X 0,Y 225.95,Z 352.748,A -85,B 0,C 180,E1 -19984.856,E2 -19984.856} C_VEL
LIN {X 0,Y 226.318,Z 346.267,A -85,B 0,C 180,E1 -19987.82,E2 -19987.82} C_VEL
LIN {X 0,Y 226.913,Z 338.34,A -85,B 0,C 180,E1 -19990.71,E2 -19990.71} C_VEL
LIN {X 0,Y 227.657,Z 329.339,A -85,B 0,C 180,E1 -19993.388,E2 -19993.388} C_VEL
LIN {X 0,Y 228.756,Z 319.245,A -85,B 0,C 180,E1 -19995.823,E2 -19995.823} C_VEL
LIN {X 0,Y 229.908,Z 307.837,A -85,B 0,C 180,E1 -19998.081,E2 -19998.081} C_VEL
LIN {X 0,Y 231.206,Z 295.808,A -85,B 0,C 180,E1 -19999.997,E2 -19999.997} C_VEL
LIN {X 0,Y 231.42,Z 290.9,A -85,B 0,C 180,E1 -20000.674,E2 -20000.674} C_VEL
LIN {X 0,Y 229.143,Z 277.537,A -85,B 0,C 180,E1 -20002.301,E2 -20002.301} C_VEL
LIN {X 0,Y 226.677,Z 262.622,A -85,B 0,C 180,E1 -20003.704,E2 -20003.704} C_VEL
LIN {X 0,Y 226.387,Z 260.287,A -85,B 0,C 180,E1 -20003.924,E2 -20003.924} C_VEL
LIN {X 0,Y 226.767,Z 260.238,A -85,B 0,C 180,E1 -20007.703,E2 -20007.703} C_VEL
LIN {X 0,Y 227.23,Z 260.18,A -85,B 0,C 180,E1 -20011.722,E2 -20011.722} C_VEL
LIN {X 0,Y 227.671,Z 260.124,A -85,B 0,C 180,E1 -20015.91,E2 -20015.91} C_VEL
LIN {X 0,Y 227.817,Z 260.106,A -85,B 0,C 180,E1 -20019.534,E2 -20019.534} C_VEL
LIN {X 0,Y 227.806,Z 260.108,A -85,B 0,C 180,E1 -20022.744,E2 -20022.744} C_VEL
LIN {X 0,Y 227.803,Z 260.108,A -85,B 0,C 180,E1 -20027.255,E2 -20027.255} C_VEL
LIN {X 0,Y 227.842,Z 260.103,A -85,B 0,C 180,E1 -20031.908,E2 -20031.908} C_VEL
LIN {X 0,Y 227.881,Z 260.1,A -85,B 0,C 180,E1 -20036.377,E2 -20036.377} C_VEL
LIN {X 0,Y 227.881,Z 260.1,A -85,B 0,C 180,E1 -20040.432,E2 -20040.432} C_VEL
LIN {X 0,Y 227.908,Z 260.097,A -85,B 0,C 180,E1 -20044.423,E2 -20044.423} C_VEL
LIN {X 0,Y 227.959,Z 260.089,A -85,B 0,C 180,E1 -20048.286,E2 -20048.286} C_VEL
LIN {X 0,Y 228.038,Z 260.075,A -85,B 0,C 180,E1 -20052.825,E2 -20052.825} C_VEL
LIN {X 0,Y 228.075,Z 260.072,A -85,B 0,C 180,E1 -20057.543,E2 -20057.543} C_VEL
LIN {X 0,Y 228.26,Z 260.053,A -85,B 0,C 180,E1 -20061.144,E2 -20061.144} C_VEL
LIN {X 0,Y 228.308,Z 260.047,A -85,B 0,C 180,E1 -20062.927,E2 -20062.927} C_VEL
LIN {X 0,Y 228.535,Z 260.019,A -85,B 0,C 180,E1 -20068.237,E2 -20068.237} C_VEL
LIN {X 0,Y 228.545,Z 260.207,A -85,B 0,C 180,E1 -20070.44,E2 -20070.44} C_VEL
LIN {X 0,Y 228.89,Z 264.679,A -85,B 0,C 180,E1 -20073.52,E2 -20073.52} C_VEL
LIN {X 0,Y 228.591,Z 270.031,A -85,B 0,C 180,E1 -20077.064,E2 -20077.064} C_VEL
LIN {X 0,Y 228.15,Z 276.928,A -85,B 0,C 180,E1 -20081.55,E2 -20081.55} C_VEL
LIN {X 0,Y 227.843,Z 281.926,A -85,B 0,C 180,E1 -20084.8,E2 -20084.8} C_VEL
LIN {X 0,Y 229.793,Z 292.267,A -85,B 0,C 180,E1 -20085.636,E2 -20085.636} C_VEL
LIN {X 0,Y 231.2,Z 301.176,A -85,B 0,C 180,E1 -20086.558,E2 -20086.558} C_VEL
LIN {X 0,Y 232.539,Z 310.923,A -85,B 0,C 180,E1 -20087.819,E2 -20087.819} C_VEL
LIN {X 0,Y 232.526,Z 314.109,A -85,B 0,C 180,E1 -20088.275,E2 -20088.275} C_VEL
LIN {X 0,Y 231.429,Z 323.033,A -85,B 0,C 180,E1 -20089.71,E2 -20089.71} C_VEL
LIN {X 0,Y 230.372,Z 330.757,A -85,B 0,C 180,E1 -20091.248,E2 -20091.248} C_VEL
LIN {X 0,Y 229.27,Z 338.439,A -85,B 0,C 180,E1 -20093.129,E2 -20093.129} C_VEL
LIN {X 0,Y 228.095,Z 346.182,A -85,B 0,C 180,E1 -20095.554,E2 -20095.554} C_VEL
LIN {X 0,Y 227.273,Z 351.382,A -85,B 0,C 180,E1 -20097.635,E2 -20097.635} C_VEL
LIN {X 0,Y 226.667,Z 355.598,A -85,B 0,C 180,E1 -20099.753,E2 -20099.753} C_VEL
LIN {X 0,Y 226.149,Z 358.911,A -85,B 0,C 180,E1 -20101.891,E2 -20101.891} C_VEL
LIN {X 0,Y 225.811,Z 361.41,A -85,B 0,C 180,E1 -20104.071,E2 -20104.071} C_VEL
LIN {X 0,Y 225.678,Z 363.112,A -85,B 0,C 180,E1 -20106.277,E2 -20106.277} C_VEL
LIN {X 0,Y 225.818,Z 364.122,A -85,B 0,C 180,E1 -20108.916,E2 -20108.916} C_VEL
LIN {X 0,Y 226.355,Z 364.021,A -85,B 0,C 180,E1 -20111.826,E2 -20111.826} C_VEL
LIN {X 0,Y 227.416,Z 361.998,A -85,B 0,C 180,E1 -20115.299,E2 -20115.299} C_VEL
LIN {X 0,Y 228.434,Z 359.587,A -85,B 0,C 180,E1 -20117.594,E2 -20117.594} C_VEL
LIN {X 0,Y 229.89,Z 355.892,A -85,B 0,C 180,E1 -20120.059,E2 -20120.059} C_VEL
LIN {X 0,Y 231.767,Z 350.516,A -85,B 0,C 180,E1 -20122.665,E2 -20122.665} C_VEL
LIN {X 0,Y 233.678,Z 344.553,A -85,B 0,C 180,E1 -20124.823,E2 -20124.823} C_VEL
LIN {X 0,Y 235.57,Z 338.216,A -85,B 0,C 180,E1 -20126.653,E2 -20126.653} C_VEL
LIN {X 0,Y 237.337,Z 331.69,A -85,B 0,C 180,E1 -20128.191,E2 -20128.191} C_VEL
LIN {X 0,Y 239.063,Z 324.374,A -85,B 0,C 180,E1 -20129.61,E2 -20129.61} C_VEL
LIN {X 0,Y 239.4,Z 320.716,A -85,B 0,C 180,E1 -20130.304,E2 -20130.304} C_VEL
LIN {X 0,Y 238.607,Z 312.135,A -85,B 0,C 180,E1 -20131.883,E2 -20131.883} C_VEL
LIN {X 0,Y 237.024,Z 303.442,A -85,B 0,C 180,E1 -20133.33,E2 -20133.33} C_VEL
LIN {X 0,Y 234.463,Z 294.035,A -85,B 0,C 180,E1 -20134.773,E2 -20134.773} C_VEL
LIN {X 0,Y 231.827,Z 286.818,A -85,B 0,C 180,E1 -20135.839,E2 -20135.839} C_VEL
LIN {X 0,Y 230.849,Z 283.906,A -85,B 0,C 180,E1 -20136.253,E2 -20136.253} C_VEL
LIN {X 0,Y 231.476,Z 278.36,A -85,B 0,C 180,E1 -20140.256,E2 -20140.256} C_VEL
LIN {X 0,Y 231.222,Z 274.619,A -85,B 0,C 180,E1 -20143.216,E2 -20143.216} C_VEL
LIN {X 0,Y 230.746,Z 271.398,A -85,B 0,C 180,E1 -20145.897,E2 -20145.897} C_VEL
